C09131=1130.125,26.875,-51.271,179.824,6.474,149.232
C09132=1130.130,26.606,-51.255,179.821,6.473,149.233
C09133=1130.135,26.356,-51.240,179.819,6.472,149.233
C09134=1130.140,26.106,-51.226,179.816,6.471,149.234
C09135=1130.145,25.857,-51.212,179.814,6.470,149.234
C09136=1130.151,25.608,-51.198,179.811,6.469,149.235
C09137=1130.156,25.358,-51.183,179.808,6.468,149.235
C09138=1130.161,25.108,-51.169,179.806,6.467,149.236
C09139=1130.166,24.859,-51.155,179.803,6.465,149.236
C09140=1130.171,24.609,-51.141,179.801,6.465,149.237
C09141=1130.176,24.360,-51.127,179.798,6.463,149.238
C09142=1130.181,24.110,-51.112,179.796,6.462,149.238
C09143=1130.186,23.860,-51.098,179.793,6.462,149.239
C09144=1130.191,23.611,-51.084,179.790,6.460,149.239
C09145=1130.197,23.362,-51.070,179.788,6.460,149.240
C09146=1130.202,23.112,-51.056,179.785,6.458,149.240
C09147=1130.207,22.862,-51.041,179.783,6.458,149.241
C09148=1130.212,22.613,-51.027,179.781,6.457,149.241
C09149=1130.217,22.364,-51.013,179.778,6.455,149.242
C09150=1130.222,22.114,-50.999,179.775,6.455,149.242
C09151=1130.227,21.864,-50.985,179.772,6.453,149.243
C09152=1130.231,21.615,-50.971,179.770,6.452,149.243
C09153=1130.237,21.366,-50.957,179.768,6.452,149.244
C09154=1130.242,21.116,-50.943,179.765,6.450,149.244
C09155=1130.247,20.866,-50.929,179.763,6.449,149.245
C09156=1130.253,20.617,-50.915,179.760,6.448,149.245
C09157=1130.258,20.367,-50.901,179.757,6.447,149.246
C09158=1130.263,20.117,-50.887,179.755,6.447,149.246
C09159=1130.267,19.868,-50.873,179.752,6.445,149.247
C09160=1130.273,19.619,-50.859,179.750,6.445,149.248
C09161=1130.278,19.369,-50.844,179.747,6.443,149.248
C09162=1130.282,19.119,-50.831,179.745,6.442,149.248
C09163=1130.288,18.870,-50.817,179.742,6.442,149.249
C09164=1130.293,18.620,-50.803,179.739,6.440,149.250
C09165=1130.298,18.370,-50.789,179.737,6.439,149.250
C09166=1130.304,18.121,-50.775,179.734,6.438,149.251
C09167=1130.308,17.872,-50.761,179.732,6.437,149.251
C09168=1130.314,17.621,-50.747,179.730,6.436,149.252
C09169=1130.319,17.373,-50.734,179.727,6.435,149.252
C09170=1130.324,17.123,-50.720,179.724,6.434,149.253
C09171=1130.328,16.873,-50.705,179.722,6.434,149.253
C09172=1130.334,16.624,-50.692,179.719,6.432,149.254
C09173=1130.339,16.374,-50.678,179.717,6.432,149.254
C09174=1130.344,16.125,-50.665,179.714,6.430,149.255
C09175=1130.349,15.875,-50.651,179.712,6.429,149.255
C09176=1130.354,15.625,-50.637,179.709,6.429,149.256
C09177=1130.360,15.376,-50.623,179.706,6.427,149.256
C09178=1130.365,15.126,-50.608,179.704,6.426,149.257
C09179=1130.369,14.876,-50.596,179.702,6.425,149.257
C09180=1130.375,14.627,-50.582,179.699,6.424,149.258
C09181=1130.380,14.377,-50.568,179.696,6.423,149.259
C09182=1130.386,14.128,-50.554,179.694,6.423,149.259
C09183=1130.390,13.879,-50.540,179.691,6.421,149.260
C09184=1130.395,13.628,-50.527,179.689,6.421,149.260
C09185=1130.401,13.379,-50.513,179.687,6.420,149.261
C09186=1130.405,13.130,-50.499,179.683,6.419,149.261
C09187=1130.411,12.880,-50.486,179.681,6.418,149.262
C09188=1130.416,12.631,-50.472,179.679,6.417,149.262
C09189=1130.422,12.381,-50.459,179.676,6.416,149.263
C09190=1130.426,12.132,-50.445,179.674,6.415,149.263
C09191=1130.431,11.881,-50.431,179.671,6.414,149.264
C09192=1130.437,11.632,-50.417,179.669,6.413,149.264
C09193=1130.441,11.383,-50.404,179.666,6.412,149.265
C09194=1130.447,11.133,-50.391,179.664,6.411,149.265
C09195=1130.452,10.883,-50.376,179.661,6.410,149.266
C09196=1130.457,10.634,-50.364,179.658,6.409,149.267
C09197=1130.462,10.384,-50.349,179.656,6.408,149.267
C09198=1130.468,10.135,-50.336,179.653,6.407,149.268
C09199=1130.472,9.885,-50.323,179.651,6.406,149.268
C09200=1130.478,9.636,-50.309,179.649,6.406,149.269
C09201=1130.483,9.386,-50.295,179.646,6.404,149.269
C09202=1130.488,9.137,-50.282,179.643,6.404,149.270
C09203=1130.493,8.887,-50.268,179.641,6.403,149.270
C09204=1130.498,8.638,-50.256,179.638,6.401,149.271
C09205=1130.503,8.387,-50.242,179.636,6.400,149.271
C09206=1130.509,8.138,-50.228,179.633,6.400,149.272
C09207=1130.513,7.888,-50.215,179.631,6.398,149.272
C09208=1130.519,7.639,-50.201,179.628,6.398,149.273
C09209=1130.523,7.389,-50.188,179.626,6.397,149.274
C09210=1130.529,7.140,-50.175,179.623,6.396,149.274
C09211=1130.533,6.890,-50.161,179.621,6.395,149.274
C09212=1130.539,6.641,-50.148,179.618,6.394,149.275
C09213=1130.544,6.391,-50.134,179.616,6.394,149.276
C09214=1130.549,6.142,-50.121,179.613,6.392,149.276
C09215=1130.555,5.891,-50.108,179.611,6.392,149.277
C09216=1130.559,5.643,-50.094,179.608,6.391,149.277
C09217=1130.565,5.392,-50.081,179.606,6.389,149.278
C09218=1130.570,5.143,-50.068,179.603,6.388,149.278
C09219=1130.575,4.894,-50.054,179.601,6.388,149.279
C09220=1130.580,4.644,-50.041,179.599,6.387,149.279
C09221=1130.586,4.394,-50.028,179.596,6.386,149.280
C09222=1130.590,4.144,-50.015,179.593,6.385,149.280
C09223=1130.596,3.895,-50.001,179.591,6.384,149.281
C09224=1130.600,3.645,-49.988,179.588,6.383,149.281
C09225=1130.606,3.396,-49.975,179.586,6.382,149.282
C09226=1130.611,3.146,-49.963,179.583,6.382,149.283
C09227=1130.616,2.897,-49.948,179.581,6.381,149.283
C09228=1130.621,2.647,-49.936,179.578,6.380,149.284
C09229=1130.626,2.397,-49.923,179.576,6.379,149.284
C09230=1130.632,2.148,-49.910,179.574,6.378,149.285
C09231=1130.637,1.899,-49.896,179.570,6.377,149.285
C09232=1130.642,1.649,-49.883,179.568,6.376,149.286
C09233=1130.647,1.380,-49.869,179.566,6.375,149.286
C09234=1130.653,1.110,-49.855,179.563,6.374,149.287
C09235=1130.659,0.840,-49.840,179.560,6.373,149.287
C09236=1130.664,0.570,-49.826,179.557,6.372,149.288
C09237=1130.670,0.321,-49.813,179.555,6.371,149.289
C09238=1130.675,0.071,-49.801,179.553,6.370,149.289
C09239=1130.680,-0.179,-49.787,179.550,6.370,149.290
C09240=1130.685,-0.428,-49.774,179.547,6.368,149.290
C09241=1130.690,-0.677,-49.761,179.545,6.367,149.291
C09242=1130.695,-0.927,-49.748,179.543,6.367,149.291
C09243=1130.700,-1.177,-49.735,179.540,6.366,149.292
C09244=1130.705,-1.426,-49.722,179.538,6.365,149.292
C09245=1130.711,-1.676,-49.709,179.535,6.364,149.293
C09246=1130.716,-1.926,-49.696,179.533,6.363,149.293
C09247=1130.721,-2.175,-49.684,179.531,6.363,149.294
C09248=1130.726,-2.425,-49.670,179.528,6.361,149.294
C09249=1130.731,-2.674,-49.657,179.525,6.361,149.295
C09250=1130.736,-2.924,-49.645,179.523,6.360,149.295
C09251=1130.742,-3.174,-49.631,179.521,6.359,149.296
C09252=1130.747,-3.423,-49.619,179.518,6.359,149.297
C09253=1130.752,-3.673,-49.606,179.515,6.357,149.297
C09254=1130.758,-3.922,-49.593,179.513,6.356,149.298
C09255=1130.762,-4.172,-49.580,179.511,6.356,149.298
C09256=1130.767,-4.422,-49.567,179.508,6.355,149.299
C09257=1130.773,-4.671,-49.555,179.506,6.353,149.299
C09258=1130.778,-4.921,-49.541,179.503,6.353,149.300
C09259=1130.783,-5.171,-49.529,179.501,6.352,149.300
C09260=1130.788,-5.420,-49.516,179.499,6.351,149.301
C09261=1130.794,-5.670,-49.503,179.496,6.351,149.301
C09262=1130.798,-5.920,-49.490,179.493,6.349,149.302
C09263=1130.804,-6.169,-49.477,179.491,6.349,149.302
C09264=1130.809,-6.418,-49.465,179.489,6.348,149.303
C09265=1130.814,-6.668,-49.452,179.486,6.347,149.304
C09266=1130.819,-6.918,-49.438,179.484,6.347,149.304
C09267=1130.824,-7.167,-49.426,179.481,6.345,149.305
C09268=1130.830,-7.417,-49.414,179.478,6.345,149.305
C09269=1130.835,-7.666,-49.401,179.476,6.344,149.306
C09270=1130.840,-7.917,-49.388,179.474,6.343,149.306
C09271=1130.845,-8.166,-49.375,179.471,6.342,149.307
C09272=1130.850,-8.415,-49.363,179.469,6.341,149.307
C09273=1130.855,-8.665,-49.350,179.467,6.340,149.308
C09274=1130.860,-8.914,-49.337,179.464,6.340,149.308
C09275=1130.865,-9.165,-49.325,179.462,6.339,149.309
C09276=1130.871,-9.414,-49.312,179.459,6.338,149.309
C09277=1130.876,-9.664,-49.299,179.457,6.337,149.310
C09278=1130.881,-9.913,-49.287,179.454,6.336,149.311
C09279=1130.887,-10.162,-49.274,179.452,6.336,149.311
C09280=1130.891,-10.413,-49.262,179.450,6.335,149.312
C09281=1130.896,-10.662,-49.249,179.447,6.334,149.312
C09282=1130.902,-10.912,-49.237,179.444,6.333,149.313
C09283=1130.907,-11.161,-49.224,179.442,6.332,149.313
C09284=1130.913,-11.411,-49.212,179.439,6.332,149.314
C09285=1130.917,-11.661,-49.199,179.437,6.331,149.314
C09286=1130.923,-11.910,-49.186,179.435,6.330,149.315
C09287=1130.928,-12.160,-49.173,179.433,6.329,149.315
C09288=1130.933,-12.410,-49.162,179.430,6.328,149.316
C09289=1130.938,-12.659,-49.149,179.427,6.327,149.316
C09290=1130.943,-12.908,-49.136,179.425,6.326,149.317
C09291=1130.948,-13.159,-49.124,179.423,6.326,149.318
C09292=1130.953,-13.408,-49.111,179.420,6.325,149.318
C09293=1130.958,-13.658,-49.099,179.418,6.324,149.319
C09294=1130.964,-13.908,-49.087,179.415,6.323,149.319
C09295=1130.969,-14.157,-49.074,179.413,6.322,149.320
C09296=1130.974,-14.406,-49.062,179.411,6.322,149.320
C09297=1130.980,-14.656,-49.050,179.408,6.321,149.321
C09298=1130.985,-14.905,-49.037,179.406,6.320,149.321
C09299=1130.989,-15.155,-49.024,179.404,6.320,149.322
C09300=1130.995,-15.406,-49.012,179.401,6.318,149.322
C09301=1131.000,-15.655,-48.999,179.398,6.318,149.323
C09302=1131.006,-15.905,-48.987,179.396,6.317,149.323
C09303=1131.011,-16.154,-48.975,179.394,6.316,149.324
C09304=1131.016,-16.404,-48.962,179.391,6.316,149.325
C09305=1131.022,-16.654,-48.950,179.389,6.315,149.325
C09306=1131.026,-16.903,-48.938,179.387,6.314,149.326
C09307=1131.031,-17.153,-48.926,179.384,6.313,149.326
C09308=1131.037,-17.402,-48.914,179.381,6.312,149.327
C09309=1131.042,-17.652,-48.902,179.379,6.311,149.327
C09310=1131.046,-17.902,-48.889,179.377,6.311,149.328
C09311=1131.052,-18.152,-48.877,179.374,6.310,149.328
C09312=1131.057,-18.401,-48.864,179.372,6.309,149.329
C09313=1131.062,-18.651,-48.853,179.370,6.309,149.329
C09314=1131.068,-18.900,-48.840,179.367,6.308,149.330
C09315=1131.073,-19.150,-48.828,179.364,6.307,149.330
C09316=1131.078,-19.400,-48.815,179.362,6.306,149.331
C09317=1131.084,-19.649,-48.804,179.360,6.305,149.331
C09318=1131.089,-19.899,-48.791,179.357,6.305,149.332
C09319=1131.094,-20.149,-48.779,179.355,6.304,149.333
C09320=1131.099,-20.398,-48.767,179.353,6.303,149.333
C09321=1131.105,-20.648,-48.755,179.350,6.303,149.334
C09322=1131.109,-20.897,-48.743,179.348,6.302,149.334
C09323=1131.114,-21.147,-48.731,179.345,6.300,149.335
C09324=1131.120,-21.397,-48.719,179.343,6.300,149.335
C09325=1131.125,-21.646,-48.706,179.341,6.299,149.336
C09326=1131.130,-21.896,-48.694,179.338,6.298,149.336
C09327=1131.136,-22.145,-48.682,179.336,6.297,149.337
C09328=1131.141,-22.395,-48.670,179.334,6.297,149.337
C09329=1131.146,-22.645,-48.658,179.331,6.296,149.338
C09330=1131.151,-22.894,-48.646,179.329,6.296,149.338
C09331=1131.156,-23.144,-48.634,179.326,6.295,149.339
C09332=1131.162,-23.394,-48.622,179.324,6.294,149.340
C09333=1131.167,-23.644,-48.610,179.322,6.293,149.340
C09334=1131.172,-23.893,-48.598,179.319,6.292,149.341
C09335=1131.178,-24.143,-48.586,179.317,6.292,149.341
C09336=1131.182,-24.392,-48.574,179.314,6.291,149.342
C09337=1131.189,-24.662,-48.561,179.312,6.290,149.342
C09338=1131.194,-24.933,-48.548,179.310,6.290,149.343
C09339=1131.199,-25.203,-48.535,179.307,6.288,149.343
C09340=1131.205,-25.473,-48.522,179.304,6.288,149.344
C09341=1131.211,-25.723,-48.510,179.302,6.287,149.345
C09342=1131.216,-25.973,-48.498,179.300,6.286,149.345
C09343=1131.221,-26.222,-48.487,179.297,6.286,149.346
C09344=1131.226,-26.472,-48.474,179.295,6.285,149.346
C09345=1131.231,-26.721,-48.463,179.293,6.284,149.347
C09346=1131.237,-26.971,-48.451,179.290,6.284,149.347
C09347=1131.241,-27.221,-48.439,179.288,6.283,149.348
C09348=1131.247,-27.470,-48.427,179.286,6.282,149.348
C09349=1131.252,-27.720,-48.415,179.282,6.281,149.349
C09350=1131.257,-27.970,-48.404,179.280,6.280,149.349
C09351=1131.263,-28.219,-48.392,179.278,6.279,149.350
C09352=1131.268,-28.469,-48.380,179.276,6.279,149.350
C09353=1131.273,-28.718,-48.368,179.273,6.278,149.351
C09354=1131.278,-28.968,-48.356,179.271,6.277,149.352
C09355=1131.283,-29.218,-48.344,179.269,6.277,149.352
C09356=1131.289,-29.468,-48.333,179.267,6.276,149.353
C09357=1131.294,-29.718,-48.321,179.264,6.275,149.353
C09358=1131.299,-29.967,-48.309,179.262,6.275,149.354
C09359=1131.304,-30.217,-48.297,179.260,6.274,149.354
C09360=1131.309,-30.466,-48.286,179.257,6.274,149.355
C09361=1131.315,-30.716,-48.274,179.255,6.273,149.355
C09362=1131.320,-30.966,-48.262,179.253,6.272,149.356
C09363=1131.325,-31.215,-48.251,179.250,6.271,149.356
C09364=1131.330,-31.465,-48.239,179.248,6.271,149.357
C09365=1131.336,-31.715,-48.227,179.246,6.270,149.357
C09366=1131.340,-31.965,-48.216,179.243,6.269,149.358
C09367=1131.346,-32.214,-48.204,179.240,6.268,149.359
C09368=1131.351,-32.464,-48.193,179.238,6.267,149.359
C09369=1131.357,-32.714,-48.181,179.236,6.266,149.360
C09370=1131.362,-32.963,-48.169,179.234,6.266,149.360
C09371=1131.367,-33.213,-48.158,179.231,6.265,149.361
C09372=1131.372,-33.463,-48.146,179.229,6.265,149.361
C09373=1131.377,-33.712,-48.135,179.227,6.264,149.362
C09374=1131.383,-33.962,-48.123,179.224,6.263,149.362
C09375=1131.388,-34.212,-48.111,179.222,6.263,149.363
C09376=1131.393,-34.461,-48.100,179.219,6.262,149.363
C09377=1131.398,-34.711,-48.088,179.217,6.261,149.364
C09378=1131.404,-34.960,-48.077,179.215,6.261,149.365
C09379=1131.409,-35.210,-48.065,179.212,6.260,149.365
C09380=1131.414,-35.460,-48.054,179.210,6.259,149.366
C09381=1131.419,-35.710,-48.042,179.208,6.258,149.366
C09382=1131.425,-35.960,-48.030,179.205,6.258,149.367
C09383=1131.430,-36.209,-48.019,179.203,6.257,149.367
C09384=1131.435,-36.459,-48.007,179.201,6.256,149.368
C09385=1131.440,-36.708,-47.996,179.198,6.256,149.368
C09386=1131.446,-36.958,-47.984,179.196,6.255,149.369
C09387=1131.451,-37.207,-47.973,179.194,6.254,149.369
C09388=1131.456,-37.457,-47.961,179.192,6.254,149.370
C09389=1131.461,-37.707,-47.951,179.189,6.253,149.370
C09390=1131.467,-37.957,-47.939,179.187,6.252,149.371
C09391=1131.472,-38.206,-47.928,179.185,6.252,149.371
C09392=1131.477,-38.456,-47.916,179.183,6.251,149.372
C09393=1131.482,-38.706,-47.905,179.180,6.251,149.373
C09394=1131.488,-38.956,-47.893,179.178,6.250,149.373
C09395=1131.493,-39.205,-47.882,179.176,6.249,149.374
C09396=1131.499,-39.455,-47.871,179.173,6.248,149.374
C09397=1131.503,-39.705,-47.860,179.171,6.248,149.375
C09398=1131.509,-39.955,-47.848,179.168,6.247,149.375
C09399=1131.514,-40.204,-47.837,179.166,6.246,149.376
C09400=1131.519,-40.453,-47.826,179.164,6.246,149.376
C09401=1131.524,-40.704,-47.814,179.161,6.245,149.377
C09402=1131.530,-40.953,-47.803,179.159,6.244,149.377
C09403=1131.535,-41.203,-47.792,179.157,6.244,149.378
C09404=1131.540,-41.452,-47.780,179.154,6.243,149.379
C09405=1131.545,-41.702,-47.768,179.152,6.242,149.379
C09406=1131.551,-41.952,-47.758,179.150,6.242,149.379
C09407=1131.556,-42.201,-47.747,179.148,6.241,149.380
C09408=1131.561,-42.451,-47.735,179.145,6.240,149.381
C09409=1131.567,-42.701,-47.725,179.143,6.240,149.381
C09410=1131.572,-42.951,-47.713,179.141,6.239,149.382
C09411=1131.577,-43.200,-47.702,179.139,6.238,149.382
C09412=1131.582,-43.449,-47.691,179.136,6.238,149.383
C09413=1131.588,-43.700,-47.679,179.134,6.237,149.383
C09414=1131.592,-43.949,-47.668,179.132,6.236,149.384
C09415=1131.598,-44.198,-47.657,179.129,6.235,149.384
C09416=1131.603,-44.449,-47.646,179.127,6.235,149.385
C09417=1131.608,-44.699,-47.635,179.125,6.234,149.385
C09418=1131.613,-44.948,-47.624,179.122,6.233,149.386
C09419=1131.619,-45.198,-47.613,179.121,6.234,149.386
C09420=1131.624,-45.448,-47.601,179.118,6.233,149.387
C09421=1131.629,-45.697,-47.591,179.116,6.232,149.388
C09422=1131.635,-45.947,-47.579,179.114,6.232,149.388
C09423=1131.640,-46.196,-47.568,179.112,6.231,149.388
C09424=1131.645,-46.446,-47.558,179.109,6.230,149.389
C09425=1131.651,-46.696,-47.546,179.107,6.230,149.390
C09426=1131.656,-46.945,-47.535,179.104,6.229,149.390
C09427=1131.661,-47.195,-47.524,179.102,6.228,149.391
C09428=1131.666,-47.445,-47.513,179.100,6.228,149.391
C09429=1131.672,-47.695,-47.502,179.097,6.227,149.392
C09430=1131.677,-47.945,-47.491,179.095,6.226,149.392
C09431=1131.682,-48.193,-47.480,179.093,6.225,149.393
C09432=1131.688,-48.444,-47.469,179.090,6.225,149.393
C09433=1131.692,-48.694,-47.458,179.088,6.224,149.394
C09434=1131.698,-48.943,-47.447,179.086,6.223,149.394
C09435=1131.703,-49.193,-47.436,179.084,6.223,149.395
C09436=1131.709,-49.443,-47.425,179.081,6.222,149.396
C09437=1131.714,-49.692,-47.414,179.080,6.222,149.396
C09438=1131.719,-49.942,-47.404,179.077,6.222,149.397
C09439=1131.724,-50.191,-47.393,179.075,6.221,149.397
C09440=1131.730,-50.442,-47.381,179.072,6.220,149.398
C09441=1131.735,-50.712,-47.370,179.070,6.220,149.398
C09442=1131.741,-50.983,-47.358,179.068,6.219,149.399
C09443=1131.747,-51.254,-47.347,179.065,6.218,149.399
C09444=1131.753,-51.525,-47.334,179.063,6.217,149.400
C09445=1131.758,-51.775,-47.323,179.060,6.217,149.401
C09446=1131.763,-52.024,-47.313,179.058,6.217,149.401
C09447=1131.768,-52.274,-47.302,179.056,6.216,149.402
C09448=1131.774,-52.523,-47.291,179.054,6.215,149.402
C09449=1131.779,-52.773,-47.281,179.052,6.214,149.403
C09450=1131.785,-53.023,-47.269,179.049,6.214,149.403
C09451=1131.790,-53.273,-47.259,179.047,6.213,149.404
C09452=1131.795,-53.522,-47.248,179.045,6.212,149.404
C09453=1131.800,-53.772,-47.237,179.043,6.212,149.405
C09454=1131.805,-54.022,-47.227,179.040,6.211,149.405
C09455=1131.810,-54.271,-47.216,179.038,6.210,149.406
C09456=1131.816,-54.521,-47.206,179.035,6.210,149.406
C09457=1131.821,-54.771,-47.194,179.034,6.210,149.407
C09458=1131.827,-55.020,-47.184,179.031,6.209,149.408
C09459=1131.832,-55.271,-47.173,179.029,6.209,149.408
C09460=1131.836,-55.520,-47.162,179.027,6.208,149.408
C09461=1131.842,-55.770,-47.151,179.025,6.207,149.409
C09462=1131.848,-56.019,-47.141,179.022,6.206,149.409
C09463=1131.853,-56.270,-47.131,179.020,6.206,149.410
C09464=1131.858,-56.518,-47.120,179.018,6.205,149.411
C09465=1131.863,-56.769,-47.109,179.015,6.204,149.411
C09466=1131.869,-57.018,-47.099,179.014,6.204,149.412
C09467=1131.873,-57.268,-47.088,179.011,6.204,149.412
C09468=1131.879,-57.517,-47.077,179.009,6.203,149.413
C09469=1131.885,-57.768,-47.066,179.007,6.202,149.413
C09470=1131.890,-58.017,-47.055,179.005,6.202,149.414
C09471=1131.895,-58.267,-47.045,179.002,6.201,149.414
C09472=1131.900,-58.517,-47.035,179.000,6.201,149.415
C09473=1131.905,-58.767,-47.024,178.998,6.200,149.415
C09474=1131.911,-59.016,-47.014,178.995,6.199,149.416
C09475=1131.916,-59.266,-47.002,178.994,6.199,149.416
C09476=1131.921,-59.516,-46.992,178.991,6.199,149.417
C09477=1131.927,-59.765,-46.982,178.989,6.198,149.418
C09478=1131.932,-60.015,-46.972,178.987,6.197,149.418
C09479=1131.937,-60.264,-46.961,178.985,6.196,149.418
C09480=1131.942,-60.515,-46.950,178.982,6.196,149.419
C09481=1131.948,-60.764,-46.940,178.980,6.195,149.420
C09482=1131.953,-61.014,-46.929,178.978,6.195,149.420
C09483=1131.958,-61.264,-46.919,178.976,6.195,149.421
C09484=1131.964,-61.513,-46.909,178.974,6.194,149.421
C09485=1131.969,-61.763,-46.898,178.971,6.193,149.422
C09486=1131.974,-62.013,-46.887,178.969,6.193,149.422
C09487=1131.979,-62.263,-46.877,178.967,6.192,149.423
C09488=1131.985,-62.512,-46.867,178.964,6.191,149.423
C09489=1131.990,-62.762,-46.857,178.963,6.191,149.424
C09490=1131.995,-63.012,-46.846,178.961,6.190,149.424
C09491=1132.000,-63.261,-46.836,178.958,6.190,149.425
C09492=1132.005,-63.512,-46.826,178.956,6.189,149.425
C09493=1132.011,-63.761,-46.815,178.954,6.188,149.426
C09494=1132.016,-64.010,-46.804,178.951,6.188,149.426
C09495=1132.021,-64.260,-46.794,178.949,6.187,149.427
C09496=1132.027,-64.510,-46.784,178.947,6.187,149.428
C09497=1132.032,-64.759,-46.773,178.945,6.187,149.428
C09498=1132.037,-65.010,-46.763,178.943,6.186,149.429
C09499=1132.043,-65.259,-46.753,178.941,6.185,149.429
C09500=1132.049,-65.509,-46.742,178.938,6.184,149.429
C09501=1132.054,-65.759,-46.732,178.936,6.184,149.430
C09502=1132.058,-66.008,-46.722,178.934,6.184,149.431
C09503=1132.063,-66.259,-46.712,178.932,6.183,149.431
C09504=1132.069,-66.508,-46.701,178.930,6.182,149.432
C09505=1132.075,-66.758,-46.691,178.928,6.182,149.432
C09506=1132.080,-67.008,-46.681,178.925,6.181,149.433
C09507=1132.085,-67.257,-46.670,178.923,6.181,149.433
C09508=1132.091,-67.507,-46.660,178.921,6.181,149.434
C09509=1132.096,-67.756,-46.651,178.919,6.180,149.434
C09510=1132.101,-68.006,-46.640,178.917,6.179,149.435
C09511=1132.106,-68.256,-46.630,178.914,6.179,149.435
C09512=1132.112,-68.505,-46.620,178.912,6.178,149.436
C09513=1132.117,-68.756,-46.609,178.910,6.177,149.436
C09514=1132.123,-69.005,-46.599,178.908,6.177,149.437
C09515=1132.127,-69.255,-46.589,178.906,6.176,149.437
C09516=1132.132,-69.505,-46.579,178.904,6.176,149.438
C09517=1132.138,-69.754,-46.568,178.901,6.175,149.439
C09518=1132.144,-70.004,-46.559,178.899,6.175,149.439
C09519=1132.149,-70.254,-46.549,178.897,6.175,149.440
C09520=1132.154,-70.504,-46.538,178.895,6.174,149.440
C09521=1132.159,-70.753,-46.529,178.893,6.173,149.441
C09522=1132.165,-71.003,-46.518,178.890,6.173,149.441
C09523=1132.171,-71.253,-46.508,178.888,6.172,149.442
C09524=1132.176,-71.503,-46.498,178.886,6.172,149.442
C09525=1132.180,-71.752,-46.488,178.884,6.171,149.443
C09526=1132.186,-72.002,-46.478,178.882,6.170,149.443
C09527=1132.191,-72.252,-46.468,178.880,6.170,149.444
C09528=1132.197,-72.502,-46.458,178.877,6.169,149.444
C09529=1132.202,-72.751,-46.448,178.876,6.169,149.445
C09530=1132.207,-73.001,-46.438,178.873,6.169,149.445
C09531=1132.213,-73.250,-46.428,178.871,6.168,149.446
C09532=1132.218,-73.501,-46.418,178.869,6.167,149.446
C09533=1132.223,-73.750,-46.408,178.867,6.166,149.447
C09534=1132.229,-74.000,-46.398,178.865,6.167,149.447
C09535=1132.234,-74.249,-46.388,178.862,6.166,149.448
C09536=1132.239,-74.500,-46.377,178.860,6.165,149.448
C09537=1132.244,-74.750,-46.368,178.858,6.164,149.449
C09538=1132.250,-74.999,-46.358,178.856,6.164,149.449
C09539=1132.256,-75.249,-46.348,178.854,6.164,149.450
C09540=1132.261,-75.498,-46.338,178.852,6.163,149.451
C09541=1132.266,-75.749,-46.328,178.849,6.163,149.451
C09542=1132.271,-75.998,-46.318,178.847,6.162,149.452
C09543=1132.277,-76.248,-46.308,178.846,6.162,149.452
C09544=1132.282,-76.497,-46.298,178.843,6.161,149.453
C09545=1132.288,-76.769,-46.288,178.841,6.161,149.453
C09546=1132.293,-77.041,-46.277,178.839,6.160,149.454
C09547=1132.299,-77.312,-46.267,178.836,6.159,149.454
C09548=1132.305,-77.583,-46.255,178.834,6.159,149.455
C09549=1132.310,-77.833,-46.246,178.831,6.158,149.455
C09550=1132.316,-78.083,-46.236,178.830,6.158,149.456
C09551=1132.321,-78.333,-46.226,178.828,6.157,149.456
C09552=1132.326,-78.583,-46.217,178.826,6.157,149.457
C09553=1132.332,-78.832,-46.206,178.823,6.156,149.457
C09554=1132.337,-79.082,-46.196,178.821,6.155,149.458
C09555=1132.343,-79.332,-46.187,178.819,6.156,149.459
C09556=1132.348,-79.581,-46.177,178.817,6.155,149.459
C09557=1132.354,-79.831,-46.167,178.815,6.154,149.459
C09558=1132.358,-80.082,-46.158,178.812,6.153,149.460
C09559=1132.364,-80.331,-46.147,178.811,6.153,149.460
C09560=1132.369,-80.581,-46.139,178.809,6.153,149.461
C09561=1132.375,-80.830,-46.128,178.806,6.152,149.461
C09562=1132.380,-81.080,-46.119,178.804,6.151,149.462
C09563=1132.385,-81.330,-46.109,178.802,6.151,149.463
C09564=1132.391,-81.579,-46.099,178.800,6.151,149.463
C09565=1132.396,-81.829,-46.090,178.798,6.150,149.464
C09566=1132.401,-82.079,-46.080,178.796,6.149,149.464
C09567=1132.406,-82.329,-46.071,178.794,6.149,149.465
C09568=1132.412,-82.579,-46.060,178.792,6.148,149.465
C09569=1132.417,-82.828,-46.051,178.789,6.148,149.466
C09570=1132.423,-83.078,-46.041,178.787,6.147,149.466
C09571=1132.428,-83.327,-46.032,178.785,6.147,149.467
C09572=1132.434,-83.578,-46.022,178.783,6.147,149.467
C09573=1132.439,-83.827,-46.012,178.781,6.146,149.468
C09574=1132.444,-84.077,-46.003,178.779,6.146,149.468
C09575=1132.449,-84.327,-45.993,178.777,6.145,149.469
C09576=1132.454,-84.577,-45.984,178.775,6.144,149.469
C09577=1132.460,-84.827,-45.973,178.772,6.144,149.470
C09578=1132.465,-85.077,-45.965,178.771,6.144,149.470
C09579=1132.471,-85.326,-45.954,178.769,6.143,149.471
C09580=1132.476,-85.576,-45.945,178.766,6.143,149.471
C09581=1132.481,-85.825,-45.936,178.764,6.142,149.472
C09582=1132.487,-86.075,-45.926,178.763,6.142,149.472
C09583=1132.492,-86.325,-45.917,178.760,6.141,149.473
C09584=1132.498,-86.575,-45.907,178.758,6.140,149.473
C09585=1132.503,-86.825,-45.898,178.756,6.141,149.474
C09586=1132.508,-87.074,-45.888,178.754,6.140,149.474
C09587=1132.513,-87.324,-45.879,178.752,6.139,149.475
C09588=1132.519,-87.574,-45.869,178.750,6.138,149.475
C09589=1132.524,-87.823,-45.860,178.748,6.139,149.476
C09590=1132.529,-88.074,-45.850,178.746,6.138,149.476
C09591=1132.534,-88.323,-45.841,178.744,6.137,149.477
C09592=1132.540,-88.573,-45.832,178.742,6.137,149.477
C09593=1132.545,-88.823,-45.822,178.740,6.136,149.478
C09594=1132.550,-89.073,-45.813,178.737,6.136,149.479
C09595=1132.556,-89.322,-45.802,178.735,6.135,149.479
C09596=1132.561,-89.572,-45.794,178.733,6.135,149.479
C09597=1132.566,-89.822,-45.785,178.731,6.134,149.480
C09598=1132.572,-90.072,-45.774,178.729,6.134,149.480
C09599=1132.577,-90.321,-45.766,178.727,6.134,149.481
C09600=1132.583,-90.572,-45.756,178.725,6.133,149.481
C09601=1132.588,-90.821,-45.746,178.723,6.132,149.482
C09602=1132.593,-91.071,-45.738,178.721,6.132,149.482
C09603=1132.599,-91.321,-45.728,178.719,6.132,149.483
C09604=1132.604,-91.570,-45.718,178.717,6.131,149.483
C09605=1132.609,-91.820,-45.710,178.715,6.131,149.484
C09606=1132.615,-92.070,-45.700,178.713,6.130,149.485
C09607=1132.620,-92.320,-45.691,178.710,6.130,149.485
C09608=1132.626,-92.569,-45.681,178.708,6.129,149.486
C09609=1132.631,-92.819,-45.672,178.707,6.129,149.486
C09610=1132.636,-93.069,-45.663,178.704,6.128,149.487
C09611=1132.641,-93.319,-45.653,178.702,6.128,149.487
C09612=1132.647,-93.569,-45.644,178.701,6.128,149.487
C09613=1132.652,-93.818,-45.635,178.698,6.127,149.488
C09614=1132.658,-94.068,-45.626,178.696,6.126,149.488
C09615=1132.663,-94.317,-45.616,178.695,6.126,149.489
C09616=1132.668,-94.567,-45.607,178.692,6.126,149.490
C09617=1132.674,-94.817,-45.598,178.690,6.125,149.490
C09618=1132.679,-95.067,-45.589,178.688,6.125,149.491
C09619=1132.685,-95.317,-45.580,178.686,6.124,149.491
C09620=1132.689,-95.566,-45.571,178.684,6.124,149.492
C09621=1132.695,-95.816,-45.561,178.682,6.124,149.492
C09622=1132.701,-96.066,-45.552,178.680,6.123,149.493
C09623=1132.706,-96.316,-45.543,178.678,6.122,149.493
C09624=1132.712,-96.566,-45.534,178.676,6.122,149.494
C09625=1132.716,-96.815,-45.524,178.674,6.121,149.494
C09626=1132.722,-97.065,-45.515,178.672,6.121,149.495
C09627=1132.727,-97.315,-45.506,178.670,6.121,149.495
C09628=1132.733,-97.564,-45.497,178.668,6.120,149.495
C09629=1132.738,-97.814,-45.488,178.666,6.119,149.496
C09630=1132.744,-98.064,-45.479,178.664,6.120,149.497
C09631=1132.749,-98.314,-45.471,178.662,6.119,149.497
C09632=1132.754,-98.564,-45.460,178.659,6.118,149.498
C09633=1132.760,-98.813,-45.451,178.658,6.118,149.498
C09634=1132.765,-99.063,-45.443,178.656,6.117,149.499
C09635=1132.770,-99.313,-45.434,178.653,6.117,149.499
C09636=1132.776,-99.563,-45.424,178.652,6.117,149.500
C09637=1132.782,-99.812,-45.416,178.650,6.116,149.500
C09638=1132.787,-100.062,-45.407,178.647,6.115,149.501
C09639=1132.792,-100.312,-45.398,178.646,6.115,149.501
C09640=1132.797,-100.562,-45.389,178.644,6.114,149.502
C09641=1132.803,-100.812,-45.379,178.641,6.114,149.502
C09642=1132.808,-101.062,-45.371,178.640,6.114,149.503
C09643=1132.813,-101.312,-45.362,178.638,6.113,149.503
C09644=1132.818,-101.562,-45.353,178.636,6.113,149.503
C09645=1132.824,-101.810,-45.344,178.634,6.112,149.504
C09646=1132.829,-102.060,-45.335,178.632,6.112,149.504
C09647=1132.835,-102.310,-45.325,178.630,6.112,149.505
C09648=1132.840,-102.560,-45.316,178.628,6.111,149.505
C09649=1132.846,-102.833,-45.307,178.625,6.111,149.506
C09650=1132.852,-103.105,-45.297,178.623,6.110,149.507
C09651=1132.857,-103.377,-45.287,178.621,6.110,149.507
C09652=1132.864,-103.649,-45.278,178.619,6.109,149.508
C09653=1132.869,-103.899,-45.269,178.617,6.108,149.508
C09654=1132.874,-104.149,-45.260,178.615,6.108,149.509
C09655=1132.879,-104.398,-45.251,178.613,6.108,149.509
C09656=1132.885,-104.649,-45.242,178.611,6.107,149.510
C09657=1132.890,-104.898,-45.233,178.609,6.107,149.510
C09658=1132.896,-105.148,-45.224,178.607,6.107,149.511
C09659=1132.901,-105.397,-45.215,178.605,6.107,149.511
C09660=1132.906,-105.647,-45.206,178.603,6.106,149.512
C09661=1132.912,-105.898,-45.198,178.601,6.105,149.512
C09662=1132.917,-106.148,-45.189,178.599,6.105,149.513
C09663=1132.923,-106.397,-45.181,178.597,6.104,149.513
C09664=1132.928,-106.647,-45.172,178.595,6.104,149.514
C09665=1132.933,-106.897,-45.163,178.593,6.104,149.514
C09666=1132.938,-107.146,-45.154,178.591,6.103,149.515
C09667=1132.943,-107.396,-45.145,178.589,6.103,149.515
C09668=1132.950,-107.646,-45.136,178.587,6.102,149.516
C09669=1132.955,-107.896,-45.127,178.585,6.102,149.516
C09670=1132.960,-108.145,-45.118,178.583,6.102,149.517
C09671=1132.966,-108.396,-45.110,178.581,6.101,149.517
C09672=1132.971,-108.645,-45.102,178.580,6.101,149.518
C09673=1132.977,-108.895,-45.093,178.577,6.100,149.518
C09674=1132.982,-109.145,-45.084,178.575,6.099,149.519
C09675=1132.987,-109.395,-45.075,178.574,6.099,149.519
C09676=1132.992,-109.644,-45.066,178.571,6.099,149.520
C09677=1132.998,-109.894,-45.057,178.570,6.099,149.520
C09678=1133.003,-110.144,-45.049,178.568,6.098,149.520
C09679=1133.009,-110.394,-45.040,178.565,6.097,149.521
C09680=1133.014,-110.644,-45.031,178.564,6.097,149.521
C09681=1133.019,-110.893,-45.023,178.562,6.097,149.522
C09682=1133.025,-111.143,-45.014,178.560,6.097,149.522
C09683=1133.030,-111.393,-45.006,178.558,6.096,149.523
C09684=1133.036,-111.642,-44.997,178.556,6.095,149.523
C09685=1133.041,-111.892,-44.988,178.554,6.095,149.524
C09686=1133.046,-112.142,-44.980,178.552,6.094,149.524
C09687=1133.051,-112.392,-44.971,178.550,6.094,149.525
C09688=1133.057,-112.642,-44.963,178.548,6.094,149.525
C09689=1133.063,-112.892,-44.954,178.546,6.094,149.526
C09690=1133.068,-113.141,-44.945,178.544,6.093,149.526
C09691=1133.074,-113.391,-44.936,178.542,6.092,149.527
C09692=1133.079,-113.641,-44.928,178.540,6.092,149.527
C09693=1133.084,-113.891,-44.919,178.538,6.092,149.528
C09694=1133.089,-114.141,-44.911,178.537,6.092,149.528
C09695=1133.095,-114.390,-44.903,178.534,6.091,149.529
C09696=1133.100,-114.640,-44.894,178.532,6.090,149.529
C09697=1133.105,-114.890,-44.885,178.531,6.090,149.530
C09698=1133.111,-115.139,-44.877,178.528,6.089,149.530
C09699=1133.116,-115.389,-44.869,178.527,6.089,149.531
C09700=1133.121,-115.639,-44.860,178.525,6.089,149.531
C09701=1133.127,-115.888,-44.851,178.523,6.089,149.532
C09702=1133.133,-116.139,-44.843,178.521,6.088,149.532
C09703=1133.138,-116.389,-44.834,178.519,6.087,149.533
C09704=1133.144,-116.638,-44.826,178.517,6.087,149.533
C09705=1133.149,-116.888,-44.818,178.515,6.086,149.533
C09706=1133.154,-117.138,-44.809,178.514,6.086,149.534
C09707=1133.160,-117.387,-44.800,178.512,6.085,149.534
C09708=1133.165,-117.638,-44.793,178.510,6.086,149.535
C09709=1133.170,-117.887,-44.784,178.508,6.085,149.535
C09710=1133.176,-118.137,-44.776,178.506,6.085,149.536
C09711=1133.181,-118.387,-44.767,178.504,6.084,149.536
C09712=1133.186,-118.637,-44.758,178.502,6.083,149.537
C09713=1133.192,-118.887,-44.750,178.500,6.083,149.537
C09714=1133.198,-119.137,-44.741,178.498,6.083,149.538
C09715=1133.202,-119.387,-44.734,178.496,6.083,149.538
C09716=1133.208,-119.636,-44.725,178.494,6.082,149.539
C09717=1133.213,-119.886,-44.716,178.493,6.082,149.539
C09718=1133.219,-120.135,-44.708,178.490,6.081,149.540
C09719=1133.224,-120.385,-44.700,178.489,6.081,149.540
C09720=1133.230,-120.636,-44.691,178.487,6.081,149.541
C09721=1133.235,-120.885,-44.683,178.484,6.080,149.541
C09722=1133.240,-121.135,-44.675,178.483,6.080,149.542
C09723=1133.246,-121.385,-44.666,178.481,6.079,149.542
C09724=1133.252,-121.635,-44.659,178.479,6.079,149.543
C09725=1133.257,-121.885,-44.650,178.477,6.078,149.543
C09726=1133.262,-122.133,-44.642,178.476,6.078,149.543
C09727=1133.267,-122.384,-44.634,178.473,6.077,149.544
C09728=1133.273,-122.634,-44.625,178.472,6.077,149.544
C09729=1133.279,-122.883,-44.617,178.470,6.077,149.545
C09730=1133.284,-123.133,-44.608,178.468,6.077,149.545
C09731=1133.289,-123.383,-44.601,178.466,6.076,149.546
C09732=1133.294,-123.633,-44.592,178.464,6.076,149.546
C09733=1133.300,-123.882,-44.584,178.462,6.075,149.547
C09734=1133.305,-124.132,-44.575,178.461,6.075,149.547
C09735=1133.310,-124.382,-44.568,178.458,6.075,149.548
C09736=1133.316,-124.632,-44.560,178.456,6.074,149.548
C09737=1133.321,-124.882,-44.551,178.455,6.074,149.549
C09738=1133.328,-125.132,-44.543,178.452,6.073,149.549
C09739=1133.332,-125.381,-44.535,178.451,6.073,149.550
C09740=1133.338,-125.631,-44.527,178.449,6.072,149.550
C09741=1133.343,-125.881,-44.518,178.447,6.072,149.551
C09742=1133.349,-126.131,-44.510,178.445,6.071,149.551
C09743=1133.354,-126.380,-44.502,178.444,6.071,149.551
C09744=1133.359,-126.631,-44.494,178.441,6.071,149.552
C09745=1133.365,-126.881,-44.486,178.440,6.071,149.552
C09746=1133.370,-127.130,-44.478,178.438,6.070,149.553
C09747=1133.376,-127.380,-44.470,178.436,6.070,149.553
C09748=1133.381,-127.630,-44.461,178.434,6.069,149.554
C09749=1133.387,-127.879,-44.453,178.432,6.069,149.554
C09750=1133.392,-128.130,-44.445,178.430,6.068,149.555
C09751=1133.398,-128.379,-44.437,178.429,6.068,149.555
C09752=1133.403,-128.629,-44.429,178.427,6.068,149.556
C09753=1132.982,-128.640,-44.473,178.423,6.072,149.557
C09754=1132.976,-128.390,-44.481,178.425,6.072,149.557
C09755=1132.971,-128.141,-44.490,178.427,6.072,149.556
C09756=1132.966,-127.891,-44.497,178.429,6.072,149.556
C09757=1132.960,-127.641,-44.506,178.431,6.073,149.556
C09758=1132.955,-127.391,-44.514,178.433,6.073,149.555
C09759=1132.949,-127.141,-44.521,178.435,6.074,149.555
C09760=1132.944,-126.892,-44.530,178.436,6.074,149.554
C09761=1132.938,-126.642,-44.538,178.438,6.075,149.554
C09762=1132.934,-126.392,-44.546,178.440,6.075,149.553
C09763=1132.928,-126.143,-44.554,178.442,6.075,149.553
C09764=1132.922,-125.892,-44.562,178.444,6.075,149.552
C09765=1132.917,-125.642,-44.571,178.446,6.076,149.552
C09766=1132.912,-125.393,-44.578,178.447,6.076,149.551
C09767=1132.906,-125.143,-44.587,178.450,6.077,149.551
C09768=1132.900,-124.893,-44.595,178.452,6.078,149.550
C09769=1132.895,-124.643,-44.604,178.453,6.078,149.550
C09770=1132.890,-124.394,-44.611,178.456,6.078,149.549
C09771=1132.885,-124.144,-44.620,178.457,6.079,149.549
C09772=1132.879,-123.894,-44.628,178.459,6.079,149.549
C09773=1132.873,-123.644,-44.637,178.460,6.079,149.548
C09774=1132.869,-123.394,-44.644,178.463,6.080,149.548
C09775=1132.863,-123.144,-44.652,178.464,6.080,149.547
C09776=1132.858,-122.895,-44.661,178.466,6.081,149.547
C09777=1132.851,-122.645,-44.669,178.468,6.081,149.546
C09778=1132.846,-122.395,-44.678,178.470,6.081,149.546
C09779=1132.842,-122.145,-44.686,178.472,6.081,149.545
C09780=1132.836,-121.896,-44.694,178.474,6.082,149.545
C09781=1132.831,-121.646,-44.703,178.476,6.082,149.544
C09782=1132.825,-121.396,-44.711,178.478,6.083,149.544
C09783=1132.820,-121.147,-44.719,178.480,6.084,149.543
C09784=1132.815,-120.896,-44.727,178.482,6.084,149.543
C09785=1132.809,-120.647,-44.736,178.483,6.085,149.543
C09786=1132.803,-120.396,-44.744,178.485,6.085,149.542
C09787=1132.798,-120.147,-44.753,178.487,6.085,149.542
C09788=1132.792,-119.897,-44.760,178.489,6.085,149.541
C09789=1132.788,-119.647,-44.769,178.491,6.086,149.541
C09790=1132.782,-119.398,-44.777,178.493,6.086,149.540
C09791=1132.776,-119.148,-44.785,178.495,6.087,149.540
C09792=1132.771,-118.898,-44.794,178.496,6.087,149.539
C09793=1132.765,-118.648,-44.802,178.499,6.087,149.539
C09794=1132.760,-118.398,-44.811,178.501,6.088,149.538
C09795=1132.755,-118.148,-44.820,178.502,6.088,149.538
C09796=1132.750,-117.899,-44.827,178.505,6.089,149.537
C09797=1132.744,-117.649,-44.836,178.506,6.089,149.537
C09798=1132.739,-117.399,-44.844,178.508,6.090,149.536
C09799=1132.733,-117.149,-44.853,178.510,6.090,149.536
C09800=1132.728,-116.900,-44.862,178.512,6.090,149.535
C09801=1132.723,-116.649,-44.870,178.514,6.090,149.535
C09802=1132.717,-116.400,-44.878,178.516,6.091,149.534
C09803=1132.712,-116.150,-44.887,178.518,6.092,149.534
C09804=1132.706,-115.900,-44.895,178.520,6.092,149.533
C09805=1132.701,-115.651,-44.903,178.522,6.092,149.533
C09806=1132.696,-115.401,-44.912,178.523,6.093,149.533
C09807=1132.690,-115.150,-44.921,178.525,6.093,149.532
C09808=1132.685,-114.901,-44.929,178.527,6.093,149.532
C09809=1132.680,-114.651,-44.938,178.529,6.094,149.531
C09810=1132.674,-114.402,-44.947,178.531,6.095,149.531
C09811=1132.668,-114.152,-44.955,178.533,6.095,149.530
C09812=1132.663,-113.902,-44.964,178.535,6.096,149.530
C09813=1132.658,-113.652,-44.972,178.537,6.096,149.529
C09814=1132.652,-113.402,-44.980,178.539,6.096,149.529
C09815=1132.647,-113.152,-44.989,178.541,6.097,149.528
C09816=1132.642,-112.903,-44.998,178.543,6.097,149.528
C09817=1132.636,-112.653,-45.007,178.545,6.098,149.527
C09818=1132.630,-112.403,-45.015,178.546,6.098,149.527
C09819=1132.625,-112.153,-45.024,178.549,6.098,149.526
C09820=1132.620,-111.903,-45.033,178.550,6.098,149.526
C09821=1132.614,-111.654,-45.041,178.552,6.099,149.525
C09822=1132.609,-111.404,-45.049,178.555,6.100,149.525
C09823=1132.604,-111.154,-45.058,178.556,6.100,149.524
C09824=1132.598,-110.904,-45.067,178.558,6.101,149.524
C09825=1132.593,-110.655,-45.076,178.560,6.101,149.523
C09826=1132.587,-110.405,-45.085,178.562,6.101,149.523
C09827=1132.582,-110.155,-45.093,178.564,6.102,149.522
C09828=1132.577,-109.905,-45.102,178.566,6.102,149.522
C09829=1132.571,-109.656,-45.110,178.568,6.103,149.521
C09830=1132.566,-109.406,-45.119,178.570,6.103,149.521
C09831=1132.561,-109.156,-45.128,178.572,6.103,149.520
C09832=1132.556,-108.906,-45.137,178.574,6.104,149.520
C09833=1132.550,-108.657,-45.145,178.576,6.104,149.519
C09834=1132.544,-108.406,-45.154,178.578,6.105,149.519
C09835=1132.539,-108.156,-45.162,178.580,6.105,149.518
C09836=1132.534,-107.907,-45.171,178.582,6.106,149.518
C09837=1132.528,-107.657,-45.180,178.584,6.106,149.517
C09838=1132.523,-107.408,-45.189,178.586,6.106,149.517
C09839=1132.518,-107.158,-45.198,178.588,6.107,149.516
C09840=1132.513,-106.908,-45.207,178.589,6.107,149.516
C09841=1132.508,-106.658,-45.215,178.592,6.108,149.515
C09842=1132.501,-106.408,-45.223,178.594,6.108,149.515
C09843=1132.496,-106.158,-45.232,178.595,6.108,149.515
C09844=1132.490,-105.908,-45.242,178.598,6.109,149.514
C09845=1132.485,-105.658,-45.251,178.600,6.110,149.514
C09846=1132.480,-105.409,-45.259,178.601,6.110,149.513
C09847=1132.474,-105.159,-45.268,178.604,6.111,149.513
C09848=1132.469,-104.910,-45.277,178.605,6.111,149.512
C09849=1132.464,-104.660,-45.286,178.607,6.111,149.512
C09850=1132.459,-104.410,-45.295,178.610,6.112,149.511
C09851=1132.454,-104.160,-45.304,178.611,6.112,149.511
C09852=1132.448,-103.910,-45.312,178.614,6.112,149.510
C09853=1132.442,-103.661,-45.322,178.616,6.113,149.509
C09854=1132.436,-103.388,-45.331,178.618,6.113,149.509
C09855=1132.431,-103.116,-45.341,178.620,6.114,149.508
C09856=1132.425,-102.844,-45.351,178.622,6.115,149.508
C09857=1132.419,-102.571,-45.360,178.624,6.115,149.507
C09858=1132.414,-102.321,-45.369,178.626,6.115,149.507
C09859=1132.409,-102.071,-45.378,178.628,6.116,149.506
C09860=1132.403,-101.822,-45.387,178.631,6.116,149.506
C09861=1132.398,-101.572,-45.396,178.632,6.116,149.505
C09862=1132.392,-101.322,-45.405,178.634,6.117,149.505
C09863=1132.387,-101.072,-45.414,178.636,6.117,149.504
C09864=1132.382,-100.823,-45.423,178.638,6.118,149.504
C09865=1132.376,-100.573,-45.432,178.640,6.119,149.503
C09866=1132.372,-100.324,-45.441,178.642,6.118,149.503
C09867=1132.365,-100.074,-45.451,178.644,6.119,149.502
C09868=1132.360,-99.824,-45.459,178.646,6.120,149.502
C09869=1132.355,-99.574,-45.468,178.648,6.120,149.501
C09870=1132.350,-99.324,-45.477,178.650,6.121,149.501
C09871=1132.344,-99.075,-45.486,178.652,6.121,149.500
C09872=1132.338,-98.824,-45.496,178.654,6.121,149.500
C09873=1132.333,-98.575,-45.504,178.656,6.122,149.499
C09874=1132.328,-98.325,-45.513,178.658,6.123,149.499
C09875=1132.323,-98.075,-45.522,178.660,6.123,149.498
C09876=1132.317,-97.826,-45.532,178.662,6.124,149.498
C09877=1132.312,-97.576,-45.541,178.664,6.124,149.498
C09878=1132.306,-97.326,-45.550,178.666,6.124,149.497
C09879=1132.301,-97.077,-45.559,178.669,6.125,149.496
C09880=1132.295,-96.826,-45.568,178.671,6.125,149.496
C09881=1132.290,-96.577,-45.577,178.672,6.125,149.495
C09882=1132.285,-96.327,-45.586,178.675,6.126,149.495
C09883=1132.279,-96.077,-45.596,178.677,6.127,149.494
C09884=1132.274,-95.827,-45.605,178.678,6.127,149.494
C09885=1132.269,-95.577,-45.614,178.681,6.128,149.493
C09886=1132.264,-95.328,-45.623,178.683,6.128,149.493
C09887=1132.258,-95.077,-45.633,178.684,6.128,149.492
C09888=1132.253,-94.829,-45.642,178.687,6.129,149.492
C09889=1132.247,-94.579,-45.651,178.689,6.130,149.491
C09890=1132.242,-94.329,-45.660,178.690,6.130,149.491
C09891=1132.236,-94.079,-45.669,178.693,6.130,149.490
C09892=1132.231,-93.830,-45.679,178.695,6.131,149.490
C09893=1132.226,-93.580,-45.688,178.697,6.131,149.489
C09894=1132.220,-93.330,-45.697,178.699,6.132,149.489
C09895=1132.215,-93.080,-45.706,178.701,6.132,149.488
C09896=1132.210,-92.830,-45.716,178.703,6.132,149.488
C09897=1132.204,-92.581,-45.725,178.705,6.133,149.487
C09898=1132.199,-92.331,-45.734,178.707,6.134,149.487
C09899=1132.193,-92.081,-45.743,178.709,6.134,149.486
C09900=1132.189,-91.831,-45.753,178.711,6.134,149.486
C09901=1132.183,-91.581,-45.762,178.713,6.135,149.485
C09902=1132.177,-91.331,-45.771,178.715,6.136,149.485
C09903=1132.173,-91.082,-45.781,178.717,6.136,149.484
C09904=1132.167,-90.832,-45.790,178.720,6.136,149.484
C09905=1132.162,-90.582,-45.799,178.722,6.137,149.483
C09906=1132.157,-90.333,-45.809,178.723,6.137,149.483
C09907=1132.151,-90.083,-45.819,178.726,6.138,149.482
C09908=1132.146,-89.833,-45.827,178.728,6.139,149.482
C09909=1132.141,-89.584,-45.837,178.729,6.138,149.481
C09910=1132.135,-89.333,-45.847,178.732,6.139,149.481
C09911=1132.130,-89.084,-45.855,178.734,6.140,149.480
C09912=1132.124,-88.834,-45.866,178.736,6.141,149.480
C09913=1132.119,-88.584,-45.875,178.738,6.141,149.479
C09914=1132.114,-88.335,-45.884,178.740,6.141,149.479
C09915=1132.108,-88.085,-45.894,178.743,6.142,149.478
C09916=1132.103,-87.835,-45.903,178.744,6.142,149.478
C09917=1132.097,-87.585,-45.913,178.746,6.143,149.477
C09918=1132.092,-87.335,-45.922,178.749,6.143,149.477
C09919=1132.087,-87.086,-45.932,178.751,6.144,149.476
C09920=1132.081,-86.836,-45.941,178.752,6.144,149.476
C09921=1132.076,-86.586,-45.950,178.754,6.145,149.475
C09922=1132.071,-86.336,-45.960,178.757,6.146,149.475
C09923=1132.066,-86.086,-45.969,178.758,6.145,149.474
C09924=1132.061,-85.837,-45.979,178.761,6.146,149.474
C09925=1132.055,-85.587,-45.988,178.763,6.147,149.473
C09926=1132.050,-85.337,-45.998,178.765,6.147,149.473
C09927=1132.045,-85.087,-46.007,178.767,6.147,149.472
C09928=1132.039,-84.838,-46.018,178.769,6.148,149.472
C09929=1132.034,-84.588,-46.026,178.771,6.149,149.471
C09930=1132.028,-84.338,-46.037,178.773,6.149,149.471
C09931=1132.023,-84.089,-46.046,178.775,6.150,149.470
C09932=1132.017,-83.839,-46.056,178.778,6.150,149.469
C09933=1132.012,-83.589,-46.065,178.780,6.151,149.469
C09934=1132.007,-83.339,-46.075,178.782,6.151,149.469
C09935=1132.002,-83.089,-46.084,178.784,6.151,149.468
C09936=1131.997,-82.840,-46.094,178.786,6.152,149.468
C09937=1131.991,-82.590,-46.103,178.788,6.153,149.467
C09938=1131.986,-82.340,-46.113,178.790,6.153,149.467
C09939=1131.980,-82.090,-46.123,178.792,6.154,149.466
C09940=1131.975,-81.841,-46.133,178.795,6.154,149.465
C09941=1131.969,-81.591,-46.143,178.797,6.155,149.465
C09942=1131.964,-81.341,-46.152,178.798,6.155,149.464
C09943=1131.959,-81.091,-46.162,178.801,6.155,149.464
C09944=1131.954,-80.841,-46.171,178.803,6.156,149.463
C09945=1131.948,-80.592,-46.181,178.805,6.157,149.463
C09946=1131.943,-80.342,-46.192,178.807,6.157,149.462
C09947=1131.938,-80.092,-46.200,178.809,6.158,149.462
C09948=1131.932,-79.843,-46.211,178.811,6.158,149.461
C09949=1131.927,-79.593,-46.220,178.814,6.159,149.461
C09950=1131.922,-79.343,-46.230,178.815,6.159,149.460
C09951=1131.916,-79.093,-46.240,178.817,6.160,149.460
C09952=1131.911,-78.843,-46.249,178.820,6.160,149.459
C09953=1131.906,-78.594,-46.259,178.822,6.161,149.459
C09954=1131.900,-78.344,-46.270,178.823,6.161,149.458
C09955=1131.895,-78.094,-46.279,178.826,6.161,149.458
C09956=1131.889,-77.845,-46.289,178.828,6.162,149.457
C09957=1131.885,-77.595,-46.299,178.830,6.163,149.457
C09958=1131.878,-77.323,-46.309,178.833,6.164,149.456
C09959=1131.873,-77.052,-46.320,178.835,6.164,149.456
C09960=1131.867,-76.780,-46.331,178.838,6.165,149.455
C09961=1131.861,-76.509,-46.342,178.839,6.165,149.455
C09962=1131.856,-76.258,-46.351,178.841,6.165,149.454
C09963=1131.851,-76.009,-46.361,178.844,6.166,149.453
C09964=1131.845,-75.760,-46.371,178.846,6.167,149.453
C09965=1131.840,-75.510,-46.381,178.848,6.167,149.452
C09966=1131.834,-75.260,-46.391,178.850,6.167,149.452
C09967=1131.829,-75.010,-46.401,178.852,6.168,149.451
C09968=1131.824,-74.760,-46.411,178.854,6.169,149.451
C09969=1131.818,-74.511,-46.421,178.857,6.169,149.450
C09970=1131.813,-74.261,-46.430,178.859,6.169,149.450
C09971=1131.807,-74.011,-46.440,178.861,6.170,149.449
C09972=1131.802,-73.761,-46.451,178.863,6.171,149.449
C09973=1131.797,-73.512,-46.461,178.865,6.171,149.448
C09974=1131.792,-73.262,-46.471,178.867,6.172,149.448
C09975=1131.786,-73.012,-46.480,178.869,6.172,149.447
C09976=1131.781,-72.762,-46.491,178.872,6.173,149.447
C09977=1131.775,-72.512,-46.501,178.874,6.173,149.446
C09978=1131.771,-72.263,-46.511,178.876,6.174,149.446
C09979=1131.765,-72.014,-46.521,178.878,6.175,149.445
C09980=1131.760,-71.763,-46.532,178.880,6.175,149.445
C09981=1131.754,-71.513,-46.541,178.883,6.175,149.444
C09982=1131.749,-71.264,-46.551,178.885,6.176,149.444
C09983=1131.744,-71.015,-46.561,178.887,6.177,149.443
C09984=1131.739,-70.764,-46.571,178.889,6.177,149.443
C09985=1131.733,-70.515,-46.582,178.891,6.177,149.442
C09986=1131.727,-70.265,-46.592,178.893,6.178,149.442
C09987=1131.723,-70.016,-46.601,178.896,6.179,149.441
C09988=1131.718,-69.766,-46.612,178.898,6.179,149.440
C09989=1131.712,-69.516,-46.622,178.900,6.180,149.440
C09990=1131.706,-69.266,-46.632,178.902,6.181,149.439
C09991=1131.701,-69.016,-46.642,178.904,6.181,149.439
C09992=1131.696,-68.767,-46.652,178.906,6.182,149.438
C09993=1131.691,-68.517,-46.662,178.909,6.182,149.438
C09994=1131.685,-68.267,-46.672,178.911,6.183,149.437
C09995=1131.680,-68.017,-46.683,178.913,6.183,149.437
C09996=1131.674,-67.768,-46.693,178.915,6.183,149.436
//INST
///DATE 2021/06/25 14:32
///ATTR SC,RW,RJ
////FRAME ROBOT
///GROUP1 RB1
NOP
MOVL C00000 V=800.0 PL=0
MOVL C00001 V=800.0 PL=0
MOVL C00002 V=800.0 PL=0
MOVL C00003 V=800.0 PL=0
MOVL C00004 V=800.0 PL=0
MOVL C00005 V=800.0 PL=0
MOVL C00006 V=800.0 PL=0
MOVL C00007 V=800.0 PL=0
MOVL C00008 V=800.0 PL=0
MOVL C00009 V=800.0 PL=0
MOVL C00010 V=800.0 PL=0
MOVL C00011 V=800.0 PL=0
MOVL C00012 V=800.0 PL=0
MOVL C00013 V=800.0 PL=0
MOVL C00014 V=800.0 PL=0
MOVL C00015 V=800.0 PL=0
MOVL C00016 V=800.0 PL=0
MOVL C00017 V=800.0 PL=0
MOVL C00018 V=800.0 PL=0
MOVL C00019 V=800.0 PL=0
MOVL C00020 V=800.0 PL=0
MOVL C00021 V=800.0 PL=0
MOVL C00022 V=800.0 PL=0
MOVL C00023 V=800.0 PL=0
MOVL C00024 V=800.0 PL=0
MOVL C00025 V=800.0 PL=0
MOVL C00026 V=800.0 PL=0
MOVL C00027 V=800.0 PL=0
MOVL C00028 V=800.0 PL=0
MOVL C00029 V=800.0 PL=0
MOVL C00030 V=800.0 PL=0
MOVL C00031 V=800.0 PL=0
MOVL C00032 V=800.0 PL=0
MOVL C00033 V=800.0 PL=0
MOVL C00034 V=800.0 PL=0
MOVL C00035 V=800.0 PL=0
MOVL C00036 V=800.0 PL=0
MOVL C00037 V=800.0 PL=0
MOVL C00038 V=800.0 PL=0
MOVL C00039 V=800.0 PL=0
MOVL C00040 V=800.0 PL=0
MOVL C00041 V=800.0 PL=0
MOVL C00042 V=800.0 PL=0
MOVL C00043 V=800.0 PL=0
MOVL C00044 V=800.0 PL=0
MOVL C00045 V=800.0 PL=0
MOVL C00046 V=800.0 PL=0
MOVL C00047 V=800.0 PL=0
MOVL C00048 V=800.0 PL=0
MOVL C00049 V=800.0 PL=0
MOVL C00050 V=800.0 PL=0
MOVL C00051 V=800.0 PL=0
MOVL C00052 V=800.0 PL=0
MOVL C00053 V=800.0 PL=0
MOVL C00054 V=800.0 PL=0
MOVL C00055 V=800.0 PL=0
MOVL C00056 V=800.0 PL=0
MOVL C00057 V=800.0 PL=0
MOVL C00058 V=800.0 PL=0
MOVL C00059 V=800.0 PL=0
MOVL C00060 V=800.0 PL=0
MOVL C00061 V=800.0 PL=0
MOVL C00062 V=800.0 PL=0
MOVL C00063 V=800.0 PL=0
MOVL C00064 V=800.0 PL=0
MOVL C00065 V=800.0 PL=0
MOVL C00066 V=800.0 PL=0
MOVL C00067 V=800.0 PL=0
MOVL C00068 V=800.0 PL=0
MOVL C00069 V=800.0 PL=0
MOVL C00070 V=800.0 PL=0
MOVL C00071 V=800.0 PL=0
MOVL C00072 V=800.0 PL=0
MOVL C00073 V=800.0 PL=0
MOVL C00074 V=800.0 PL=0
MOVL C00075 V=800.0 PL=0
MOVL C00076 V=800.0 PL=0
MOVL C00077 V=800.0 PL=0
MOVL C00078 V=800.0 PL=0
MOVL C00079 V=800.0 PL=0
MOVL C00080 V=800.0 PL=0
MOVL C00081 V=800.0 PL=0
MOVL C00082 V=800.0 PL=0
MOVL C00083 V=800.0 PL=0
MOVL C00084 V=800.0 PL=0
MOVL C00085 V=800.0 PL=0
MOVL C00086 V=800.0 PL=0
MOVL C00087 V=800.0 PL=0
MOVL C00088 V=800.0 PL=0
MOVL C00089 V=800.0 PL=0
MOVL C00090 V=800.0 PL=0
MOVL C00091 V=800.0 PL=0
MOVL C00092 V=800.0 PL=0
MOVL C00093 V=800.0 PL=0
MOVL C00094 V=800.0 PL=0
MOVL C00095 V=800.0 PL=0
MOVL C00096 V=800.0 PL=0
MOVL C00097 V=800.0 PL=0
MOVL C00098 V=800.0 PL=0
MOVL C00099 V=800.0 PL=0
MOVL C00100 V=800.0 PL=0
MOVL C00101 V=800.0 PL=0
MOVL C00102 V=800.0 PL=0
MOVL C00103 V=800.0 PL=0
MOVL C00104 V=800.0 PL=0
MOVL C00105 V=800.0 PL=0
MOVL C00106 V=800.0 PL=0
MOVL C00107 V=800.0 PL=0
MOVL C00108 V=800.0 PL=0
MOVL C00109 V=800.0 PL=0
MOVL C00110 V=800.0 PL=0
MOVL C00111 V=800.0 PL=0
MOVL C00112 V=800.0 PL=0
MOVL C00113 V=800.0 PL=0
MOVL C00114 V=800.0 PL=0
MOVL C00115 V=800.0 PL=0
MOVL C00116 V=800.0 PL=0
MOVL C00117 V=800.0 PL=0
MOVL C00118 V=800.0 PL=0
MOVL C00119 V=800.0 PL=0
MOVL C00120 V=800.0 PL=0
MOVL C00121 V=800.0 PL=0
MOVL C00122 V=800.0 PL=0
MOVL C00123 V=800.0 PL=0
MOVL C00124 V=800.0 PL=0
MOVL C00125 V=800.0 PL=0
MOVL C00126 V=800.0 PL=0
MOVL C00127 V=800.0 PL=0
MOVL C00128 V=800.0 PL=0
MOVL C00129 V=800.0 PL=0
MOVL C00130 V=800.0 PL=0
MOVL C00131 V=800.0 PL=0
MOVL C00132 V=800.0 PL=0
MOVL C00133 V=800.0 PL=0
MOVL C00134 V=800.0 PL=0
MOVL C00135 V=800.0 PL=0
MOVL C00136 V=800.0 PL=0
MOVL C00137 V=800.0 PL=0
MOVL C00138 V=800.0 PL=0
MOVL C00139 V=800.0 PL=0
MOVL C00140 V=800.0 PL=0
MOVL C00141 V=800.0 PL=0
MOVL C00142 V=800.0 PL=0
MOVL C00143 V=800.0 PL=0
MOVL C00144 V=800.0 PL=0
MOVL C00145 V=800.0 PL=0
MOVL C00146 V=800.0 PL=0
MOVL C00147 V=800.0 PL=0
MOVL C00148 V=800.0 PL=0
MOVL C00149 V=800.0 PL=0
MOVL C00150 V=800.0 PL=0
MOVL C00151 V=800.0 PL=0
MOVL C00152 V=800.0 PL=0
MOVL C00153 V=800.0 PL=0
MOVL C00154 V=800.0 PL=0
MOVL C00155 V=800.0 PL=0
MOVL C00156 V=800.0 PL=0
MOVL C00157 V=800.0 PL=0
MOVL C00158 V=800.0 PL=0
MOVL C00159 V=800.0 PL=0
MOVL C00160 V=800.0 PL=0
MOVL C00161 V=800.0 PL=0
MOVL C00162 V=800.0 PL=0
MOVL C00163 V=800.0 PL=0
MOVL C00164 V=800.0 PL=0
MOVL C00165 V=800.0 PL=0
MOVL C00166 V=800.0 PL=0
MOVL C00167 V=800.0 PL=0
MOVL C00168 V=800.0 PL=0
MOVL C00169 V=800.0 PL=0
MOVL C00170 V=800.0 PL=0
MOVL C00171 V=800.0 PL=0
MOVL C00172 V=800.0 PL=0
MOVL C00173 V=800.0 PL=0
MOVL C00174 V=800.0 PL=0
MOVL C00175 V=800.0 PL=0
MOVL C00176 V=800.0 PL=0
MOVL C00177 V=800.0 PL=0
MOVL C00178 V=800.0 PL=0
MOVL C00179 V=800.0 PL=0
MOVL C00180 V=800.0 PL=0
MOVL C00181 V=800.0 PL=0
MOVL C00182 V=800.0 PL=0
MOVL C00183 V=800.0 PL=0
MOVL C00184 V=800.0 PL=0
MOVL C00185 V=800.0 PL=0
MOVL C00186 V=800.0 PL=0
MOVL C00187 V=800.0 PL=0
MOVL C00188 V=800.0 PL=0
MOVL C00189 V=800.0 PL=0
MOVL C00190 V=800.0 PL=0
MOVL C00191 V=800.0 PL=0
MOVL C00192 V=800.0 PL=0
MOVL C00193 V=800.0 PL=0
MOVL C00194 V=800.0 PL=0
MOVL C00195 V=800.0 PL=0
MOVL C00196 V=800.0 PL=0
MOVL C00197 V=800.0 PL=0
MOVL C00198 V=800.0 PL=0
MOVL C00199 V=800.0 PL=0
MOVL C00200 V=800.0 PL=0
MOVL C00201 V=800.0 PL=0
MOVL C00202 V=800.0 PL=0
MOVL C00203 V=800.0 PL=0
MOVL C00204 V=800.0 PL=0
MOVL C00205 V=800.0 PL=0
MOVL C00206 V=800.0 PL=0
MOVL C00207 V=800.0 PL=0
MOVL C00208 V=800.0 PL=0
MOVL C00209 V=800.0 PL=0
MOVL C00210 V=800.0 PL=0
MOVL C00211 V=800.0 PL=0
MOVL C00212 V=800.0 PL=0
MOVL C00213 V=800.0 PL=0
MOVL C00214 V=800.0 PL=0
MOVL C00215 V=800.0 PL=0
MOVL C00216 V=800.0 PL=0
MOVL C00217 V=800.0 PL=0
MOVL C00218 V=800.0 PL=0
MOVL C00219 V=800.0 PL=0
MOVL C00220 V=800.0 PL=0
MOVL C00221 V=800.0 PL=0
MOVL C00222 V=800.0 PL=0
MOVL C00223 V=800.0 PL=0
MOVL C00224 V=800.0 PL=0
MOVL C00225 V=800.0 PL=0
MOVL C00226 V=800.0 PL=0
MOVL C00227 V=800.0 PL=0
MOVL C00228 V=800.0 PL=0
MOVL C00229 V=800.0 PL=0
MOVL C00230 V=800.0 PL=0
MOVL C00231 V=800.0 PL=0
MOVL C00232 V=800.0 PL=0
MOVL C00233 V=800.0 PL=0
MOVL C00234 V=800.0 PL=0
MOVL C00235 V=800.0 PL=0
MOVL C00236 V=800.0 PL=0
MOVL C00237 V=800.0 PL=0
MOVL C00238 V=800.0 PL=0
MOVL C00239 V=800.0 PL=0
MOVL C00240 V=800.0 PL=0
MOVL C00241 V=800.0 PL=0
MOVL C00242 V=800.0 PL=0
MOVL C00243 V=800.0 PL=0
MOVL C00244 V=800.0 PL=0
MOVL C00245 V=800.0 PL=0
MOVL C00246 V=800.0 PL=0
MOVL C00247 V=800.0 PL=0
MOVL C00248 V=800.0 PL=0
MOVL C00249 V=800.0 PL=0
MOVL C00250 V=800.0 PL=0
MOVL C00251 V=800.0 PL=0
MOVL C00252 V=800.0 PL=0
MOVL C00253 V=800.0 PL=0
MOVL C00254 V=800.0 PL=0
MOVL C00255 V=800.0 PL=0
MOVL C00256 V=800.0 PL=0
MOVL C00257 V=800.0 PL=0
MOVL C00258 V=800.0 PL=0
MOVL C00259 V=800.0 PL=0
MOVL C00260 V=800.0 PL=0
MOVL C00261 V=800.0 PL=0
MOVL C00262 V=800.0 PL=0
MOVL C00263 V=800.0 PL=0
MOVL C00264 V=800.0 PL=0
MOVL C00265 V=800.0 PL=0
MOVL C00266 V=800.0 PL=0
MOVL C00267 V=800.0 PL=0
MOVL C00268 V=800.0 PL=0
MOVL C00269 V=800.0 PL=0
MOVL C00270 V=800.0 PL=0
MOVL C00271 V=800.0 PL=0
MOVL C00272 V=800.0 PL=0
MOVL C00273 V=800.0 PL=0
MOVL C00274 V=800.0 PL=0
MOVL C00275 V=800.0 PL=0
MOVL C00276 V=800.0 PL=0
MOVL C00277 V=800.0 PL=0
MOVL C00278 V=800.0 PL=0
MOVL C00279 V=800.0 PL=0
MOVL C00280 V=800.0 PL=0
MOVL C00281 V=800.0 PL=0
MOVL C00282 V=800.0 PL=0
MOVL C00283 V=800.0 PL=0
MOVL C00284 V=800.0 PL=0
MOVL C00285 V=800.0 PL=0
MOVL C00286 V=800.0 PL=0
MOVL C00287 V=800.0 PL=0
MOVL C00288 V=800.0 PL=0
MOVL C00289 V=800.0 PL=0
MOVL C00290 V=800.0 PL=0
MOVL C00291 V=800.0 PL=0
MOVL C00292 V=800.0 PL=0
MOVL C00293 V=800.0 PL=0
MOVL C00294 V=800.0 PL=0
MOVL C00295 V=800.0 PL=0
MOVL C00296 V=800.0 PL=0
MOVL C00297 V=800.0 PL=0
MOVL C00298 V=800.0 PL=0
MOVL C00299 V=800.0 PL=0
MOVL C00300 V=800.0 PL=0
MOVL C00301 V=800.0 PL=0
MOVL C00302 V=800.0 PL=0
MOVL C00303 V=800.0 PL=0
MOVL C00304 V=800.0 PL=0
MOVL C00305 V=800.0 PL=0
MOVL C00306 V=800.0 PL=0
MOVL C00307 V=800.0 PL=0
MOVL C00308 V=800.0 PL=0
MOVL C00309 V=800.0 PL=0
MOVL C00310 V=800.0 PL=0
MOVL C00311 V=800.0 PL=0
MOVL C00312 V=800.0 PL=0
MOVL C00313 V=800.0 PL=0
MOVL C00314 V=800.0 PL=0
MOVL C00315 V=800.0 PL=0
MOVL C00316 V=800.0 PL=0
MOVL C00317 V=800.0 PL=0
MOVL C00318 V=800.0 PL=0
MOVL C00319 V=800.0 PL=0
MOVL C00320 V=800.0 PL=0
MOVL C00321 V=800.0 PL=0
MOVL C00322 V=800.0 PL=0
MOVL C00323 V=800.0 PL=0
MOVL C00324 V=800.0 PL=0
MOVL C00325 V=800.0 PL=0
MOVL C00326 V=800.0 PL=0
MOVL C00327 V=800.0 PL=0
MOVL C00328 V=800.0 PL=0
MOVL C00329 V=800.0 PL=0
MOVL C00330 V=800.0 PL=0
MOVL C00331 V=800.0 PL=0
MOVL C00332 V=800.0 PL=0
MOVL C00333 V=800.0 PL=0
MOVL C00334 V=800.0 PL=0
MOVL C00335 V=800.0 PL=0
MOVL C00336 V=800.0 PL=0
MOVL C00337 V=800.0 PL=0
MOVL C00338 V=800.0 PL=0
MOVL C00339 V=800.0 PL=0
MOVL C00340 V=800.0 PL=0
MOVL C00341 V=800.0 PL=0
MOVL C00342 V=800.0 PL=0
MOVL C00343 V=800.0 PL=0
MOVL C00344 V=800.0 PL=0
MOVL C00345 V=800.0 PL=0
MOVL C00346 V=800.0 PL=0
MOVL C00347 V=800.0 PL=0
MOVL C00348 V=800.0 PL=0
MOVL C00349 V=800.0 PL=0
MOVL C00350 V=800.0 PL=0
MOVL C00351 V=800.0 PL=0
MOVL C00352 V=800.0 PL=0
MOVL C00353 V=800.0 PL=0
MOVL C00354 V=800.0 PL=0
MOVL C00355 V=800.0 PL=0
MOVL C00356 V=800.0 PL=0
MOVL C00357 V=800.0 PL=0
MOVL C00358 V=800.0 PL=0
MOVL C00359 V=800.0 PL=0
MOVL C00360 V=800.0 PL=0
MOVL C00361 V=800.0 PL=0
MOVL C00362 V=800.0 PL=0
MOVL C00363 V=800.0 PL=0
MOVL C00364 V=800.0 PL=0
MOVL C00365 V=800.0 PL=0
MOVL C00366 V=800.0 PL=0
MOVL C00367 V=800.0 PL=0
MOVL C00368 V=800.0 PL=0
MOVL C00369 V=800.0 PL=0
MOVL C00370 V=800.0 PL=0
MOVL C00371 V=800.0 PL=0
MOVL C00372 V=800.0 PL=0
MOVL C00373 V=800.0 PL=0
MOVL C00374 V=800.0 PL=0
MOVL C00375 V=800.0 PL=0
MOVL C00376 V=800.0 PL=0
MOVL C00377 V=800.0 PL=0
MOVL C00378 V=800.0 PL=0
MOVL C00379 V=800.0 PL=0
MOVL C00380 V=800.0 PL=0
MOVL C00381 V=800.0 PL=0
MOVL C00382 V=800.0 PL=0
MOVL C00383 V=800.0 PL=0
MOVL C00384 V=800.0 PL=0
MOVL C00385 V=800.0 PL=0
MOVL C00386 V=800.0 PL=0
MOVL C00387 V=800.0 PL=0
MOVL C00388 V=800.0 PL=0
MOVL C00389 V=800.0 PL=0
MOVL C00390 V=800.0 PL=0
MOVL C00391 V=800.0 PL=0
MOVL C00392 V=800.0 PL=0
MOVL C00393 V=800.0 PL=0
MOVL C00394 V=800.0 PL=0
MOVL C00395 V=800.0 PL=0
MOVL C00396 V=800.0 PL=0
MOVL C00397 V=800.0 PL=0
MOVL C00398 V=800.0 PL=0
MOVL C00399 V=800.0 PL=0
MOVL C00400 V=800.0 PL=0
MOVL C00401 V=800.0 PL=0
MOVL C00402 V=800.0 PL=0
MOVL C00403 V=800.0 PL=0
MOVL C00404 V=800.0 PL=0
MOVL C00405 V=800.0 PL=0
MOVL C00406 V=800.0 PL=0
MOVL C00407 V=800.0 PL=0
MOVL C00408 V=800.0 PL=0
MOVL C00409 V=800.0 PL=0
MOVL C00410 V=800.0 PL=0
MOVL C00411 V=800.0 PL=0
MOVL C00412 V=800.0 PL=0
MOVL C00413 V=800.0 PL=0
MOVL C00414 V=800.0 PL=0
MOVL C00415 V=800.0 PL=0
MOVL C00416 V=800.0 PL=0
MOVL C00417 V=800.0 PL=0
MOVL C00418 V=800.0 PL=0
MOVL C00419 V=800.0 PL=0
MOVL C00420 V=800.0 PL=0
MOVL C00421 V=800.0 PL=0
MOVL C00422 V=800.0 PL=0
MOVL C00423 V=800.0 PL=0
MOVL C00424 V=800.0 PL=0
MOVL C00425 V=800.0 PL=0
MOVL C00426 V=800.0 PL=0
MOVL C00427 V=800.0 PL=0
MOVL C00428 V=800.0 PL=0
MOVL C00429 V=800.0 PL=0
MOVL C00430 V=800.0 PL=0
MOVL C00431 V=800.0 PL=0
MOVL C00432 V=800.0 PL=0
MOVL C00433 V=800.0 PL=0
MOVL C00434 V=800.0 PL=0
MOVL C00435 V=800.0 PL=0
MOVL C00436 V=800.0 PL=0
MOVL C00437 V=800.0 PL=0
MOVL C00438 V=800.0 PL=0
MOVL C00439 V=800.0 PL=0
MOVL C00440 V=800.0 PL=0
MOVL C00441 V=800.0 PL=0
MOVL C00442 V=800.0 PL=0
MOVL C00443 V=800.0 PL=0
MOVL C00444 V=800.0 PL=0
MOVL C00445 V=800.0 PL=0
MOVL C00446 V=800.0 PL=0
MOVL C00447 V=800.0 PL=0
MOVL C00448 V=800.0 PL=0
MOVL C00449 V=800.0 PL=0
MOVL C00450 V=800.0 PL=0
MOVL C00451 V=800.0 PL=0
MOVL C00452 V=800.0 PL=0
MOVL C00453 V=800.0 PL=0
MOVL C00454 V=800.0 PL=0
MOVL C00455 V=800.0 PL=0
MOVL C00456 V=800.0 PL=0
MOVL C00457 V=800.0 PL=0
MOVL C00458 V=800.0 PL=0
MOVL C00459 V=800.0 PL=0
MOVL C00460 V=800.0 PL=0
MOVL C00461 V=800.0 PL=0
MOVL C00462 V=800.0 PL=0
MOVL C00463 V=800.0 PL=0
MOVL C00464 V=800.0 PL=0
MOVL C00465 V=800.0 PL=0
MOVL C00466 V=800.0 PL=0
MOVL C00467 V=800.0 PL=0
MOVL C00468 V=800.0 PL=0
MOVL C00469 V=800.0 PL=0
MOVL C00470 V=800.0 PL=0
MOVL C00471 V=800.0 PL=0
MOVL C00472 V=800.0 PL=0
MOVL C00473 V=800.0 PL=0
MOVL C00474 V=800.0 PL=0
MOVL C00475 V=800.0 PL=0
MOVL C00476 V=800.0 PL=0
MOVL C00477 V=800.0 PL=0
MOVL C00478 V=800.0 PL=0
MOVL C00479 V=800.0 PL=0
MOVL C00480 V=800.0 PL=0
MOVL C00481 V=800.0 PL=0
MOVL C00482 V=800.0 PL=0
MOVL C00483 V=800.0 PL=0
MOVL C00484 V=800.0 PL=0
MOVL C00485 V=800.0 PL=0
MOVL C00486 V=800.0 PL=0
MOVL C00487 V=800.0 PL=0
MOVL C00488 V=800.0 PL=0
MOVL C00489 V=800.0 PL=0
MOVL C00490 V=800.0 PL=0
MOVL C00491 V=800.0 PL=0
MOVL C00492 V=800.0 PL=0
MOVL C00493 V=800.0 PL=0
MOVL C00494 V=800.0 PL=0
MOVL C00495 V=800.0 PL=0
MOVL C00496 V=800.0 PL=0
MOVL C00497 V=800.0 PL=0
MOVL C00498 V=800.0 PL=0
MOVL C00499 V=800.0 PL=0
MOVL C00500 V=800.0 PL=0
MOVL C00501 V=800.0 PL=0
MOVL C00502 V=800.0 PL=0
MOVL C00503 V=800.0 PL=0
MOVL C00504 V=800.0 PL=0
MOVL C00505 V=800.0 PL=0
MOVL C00506 V=800.0 PL=0
MOVL C00507 V=800.0 PL=0
MOVL C00508 V=800.0 PL=0
MOVL C00509 V=800.0 PL=0
MOVL C00510 V=800.0 PL=0
MOVL C00511 V=800.0 PL=0
MOVL C00512 V=800.0 PL=0
MOVL C00513 V=800.0 PL=0
MOVL C00514 V=800.0 PL=0
MOVL C00515 V=800.0 PL=0
MOVL C00516 V=800.0 PL=0
MOVL C00517 V=800.0 PL=0
MOVL C00518 V=800.0 PL=0
MOVL C00519 V=800.0 PL=0
MOVL C00520 V=800.0 PL=0
MOVL C00521 V=800.0 PL=0
MOVL C00522 V=800.0 PL=0
MOVL C00523 V=800.0 PL=0
MOVL C00524 V=800.0 PL=0
MOVL C00525 V=800.0 PL=0
MOVL C00526 V=800.0 PL=0
MOVL C00527 V=800.0 PL=0
MOVL C00528 V=800.0 PL=0
MOVL C00529 V=800.0 PL=0
MOVL C00530 V=800.0 PL=0
MOVL C00531 V=800.0 PL=0
MOVL C00532 V=800.0 PL=0
MOVL C00533 V=800.0 PL=0
MOVL C00534 V=800.0 PL=0
MOVL C00535 V=800.0 PL=0
MOVL C00536 V=800.0 PL=0
MOVL C00537 V=800.0 PL=0
MOVL C00538 V=800.0 PL=0
MOVL C00539 V=800.0 PL=0
MOVL C00540 V=800.0 PL=0
MOVL C00541 V=800.0 PL=0
MOVL C00542 V=800.0 PL=0
MOVL C00543 V=800.0 PL=0
MOVL C00544 V=800.0 PL=0
MOVL C00545 V=800.0 PL=0
MOVL C00546 V=800.0 PL=0
MOVL C00547 V=800.0 PL=0
MOVL C00548 V=800.0 PL=0
MOVL C00549 V=800.0 PL=0
MOVL C00550 V=800.0 PL=0
MOVL C00551 V=800.0 PL=0
MOVL C00552 V=800.0 PL=0
MOVL C00553 V=800.0 PL=0
MOVL C00554 V=800.0 PL=0
MOVL C00555 V=800.0 PL=0
MOVL C00556 V=800.0 PL=0
MOVL C00557 V=800.0 PL=0
MOVL C00558 V=800.0 PL=0
MOVL C00559 V=800.0 PL=0
MOVL C00560 V=800.0 PL=0
MOVL C00561 V=800.0 PL=0
MOVL C00562 V=800.0 PL=0
MOVL C00563 V=800.0 PL=0
MOVL C00564 V=800.0 PL=0
MOVL C00565 V=800.0 PL=0
MOVL C00566 V=800.0 PL=0
MOVL C00567 V=800.0 PL=0
MOVL C00568 V=800.0 PL=0
MOVL C00569 V=800.0 PL=0
MOVL C00570 V=800.0 PL=0
MOVL C00571 V=800.0 PL=0
MOVL C00572 V=800.0 PL=0
MOVL C00573 V=800.0 PL=0
MOVL C00574 V=800.0 PL=0
MOVL C00575 V=800.0 PL=0
MOVL C00576 V=800.0 PL=0
MOVL C00577 V=800.0 PL=0
MOVL C00578 V=800.0 PL=0
MOVL C00579 V=800.0 PL=0
MOVL C00580 V=800.0 PL=0
MOVL C00581 V=800.0 PL=0
MOVL C00582 V=800.0 PL=0
MOVL C00583 V=800.0 PL=0
MOVL C00584 V=800.0 PL=0
MOVL C00585 V=800.0 PL=0
MOVL C00586 V=800.0 PL=0
MOVL C00587 V=800.0 PL=0
MOVL C00588 V=800.0 PL=0
MOVL C00589 V=800.0 PL=0
MOVL C00590 V=800.0 PL=0
MOVL C00591 V=800.0 PL=0
MOVL C00592 V=800.0 PL=0
MOVL C00593 V=800.0 PL=0
MOVL C00594 V=800.0 PL=0
MOVL C00595 V=800.0 PL=0
MOVL C00596 V=800.0 PL=0
MOVL C00597 V=800.0 PL=0
MOVL C00598 V=800.0 PL=0
MOVL C00599 V=800.0 PL=0
MOVL C00600 V=800.0 PL=0
MOVL C00601 V=800.0 PL=0
MOVL C00602 V=800.0 PL=0
MOVL C00603 V=800.0 PL=0
MOVL C00604 V=800.0 PL=0
MOVL C00605 V=800.0 PL=0
MOVL C00606 V=800.0 PL=0
MOVL C00607 V=800.0 PL=0
MOVL C00608 V=800.0 PL=0
MOVL C00609 V=800.0 PL=0
MOVL C00610 V=800.0 PL=0
MOVL C00611 V=800.0 PL=0
MOVL C00612 V=800.0 PL=0
MOVL C00613 V=800.0 PL=0
MOVL C00614 V=800.0 PL=0
MOVL C00615 V=800.0 PL=0
MOVL C00616 V=800.0 PL=0
MOVL C00617 V=800.0 PL=0
MOVL C00618 V=800.0 PL=0
MOVL C00619 V=800.0 PL=0
MOVL C00620 V=800.0 PL=0
MOVL C00621 V=800.0 PL=0
MOVL C00622 V=800.0 PL=0
MOVL C00623 V=800.0 PL=0
MOVL C00624 V=800.0 PL=0
MOVL C00625 V=800.0 PL=0
MOVL C00626 V=800.0 PL=0
MOVL C00627 V=800.0 PL=0
MOVL C00628 V=800.0 PL=0
MOVL C00629 V=800.0 PL=0
MOVL C00630 V=800.0 PL=0
MOVL C00631 V=800.0 PL=0
MOVL C00632 V=800.0 PL=0
MOVL C00633 V=800.0 PL=0
MOVL C00634 V=800.0 PL=0
MOVL C00635 V=800.0 PL=0
MOVL C00636 V=800.0 PL=0
MOVL C00637 V=800.0 PL=0
MOVL C00638 V=800.0 PL=0
MOVL C00639 V=800.0 PL=0
MOVL C00640 V=800.0 PL=0
MOVL C00641 V=800.0 PL=0
MOVL C00642 V=800.0 PL=0
MOVL C00643 V=800.0 PL=0
MOVL C00644 V=800.0 PL=0
MOVL C00645 V=800.0 PL=0
MOVL C00646 V=800.0 PL=0
MOVL C00647 V=800.0 PL=0
MOVL C00648 V=800.0 PL=0
MOVL C00649 V=800.0 PL=0
MOVL C00650 V=800.0 PL=0
MOVL C00651 V=800.0 PL=0
MOVL C00652 V=800.0 PL=0
MOVL C00653 V=800.0 PL=0
MOVL C00654 V=800.0 PL=0
MOVL C00655 V=800.0 PL=0
MOVL C00656 V=800.0 PL=0
MOVL C00657 V=800.0 PL=0
MOVL C00658 V=800.0 PL=0
MOVL C00659 V=800.0 PL=0
MOVL C00660 V=800.0 PL=0
MOVL C00661 V=800.0 PL=0
MOVL C00662 V=800.0 PL=0
MOVL C00663 V=800.0 PL=0
MOVL C00664 V=800.0 PL=0
MOVL C00665 V=800.0 PL=0
MOVL C00666 V=800.0 PL=0
MOVL C00667 V=800.0 PL=0
MOVL C00668 V=800.0 PL=0
MOVL C00669 V=800.0 PL=0
MOVL C00670 V=800.0 PL=0
MOVL C00671 V=800.0 PL=0
MOVL C00672 V=800.0 PL=0
MOVL C00673 V=800.0 PL=0
MOVL C00674 V=800.0 PL=0
MOVL C00675 V=800.0 PL=0
MOVL C00676 V=800.0 PL=0
MOVL C00677 V=800.0 PL=0
MOVL C00678 V=800.0 PL=0
MOVL C00679 V=800.0 PL=0
MOVL C00680 V=800.0 PL=0
MOVL C00681 V=800.0 PL=0
MOVL C00682 V=800.0 PL=0
MOVL C00683 V=800.0 PL=0
MOVL C00684 V=800.0 PL=0
MOVL C00685 V=800.0 PL=0
MOVL C00686 V=800.0 PL=0
MOVL C00687 V=800.0 PL=0
MOVL C00688 V=800.0 PL=0
MOVL C00689 V=800.0 PL=0
MOVL C00690 V=800.0 PL=0
MOVL C00691 V=800.0 PL=0
MOVL C00692 V=800.0 PL=0
MOVL C00693 V=800.0 PL=0
MOVL C00694 V=800.0 PL=0
MOVL C00695 V=800.0 PL=0
MOVL C00696 V=800.0 PL=0
MOVL C00697 V=800.0 PL=0
MOVL C00698 V=800.0 PL=0
MOVL C00699 V=800.0 PL=0
MOVL C00700 V=800.0 PL=0
MOVL C00701 V=800.0 PL=0
MOVL C00702 V=800.0 PL=0
MOVL C00703 V=800.0 PL=0
MOVL C00704 V=800.0 PL=0
MOVL C00705 V=800.0 PL=0
MOVL C00706 V=800.0 PL=0
MOVL C00707 V=800.0 PL=0
MOVL C00708 V=800.0 PL=0
MOVL C00709 V=800.0 PL=0
MOVL C00710 V=800.0 PL=0
MOVL C00711 V=800.0 PL=0
MOVL C00712 V=800.0 PL=0
MOVL C00713 V=800.0 PL=0
MOVL C00714 V=800.0 PL=0
MOVL C00715 V=800.0 PL=0
MOVL C00716 V=800.0 PL=0
MOVL C00717 V=800.0 PL=0
MOVL C00718 V=800.0 PL=0
MOVL C00719 V=800.0 PL=0
MOVL C00720 V=800.0 PL=0
MOVL C00721 V=800.0 PL=0
MOVL C00722 V=800.0 PL=0
MOVL C00723 V=800.0 PL=0
MOVL C00724 V=800.0 PL=0
MOVL C00725 V=800.0 PL=0
MOVL C00726 V=800.0 PL=0
MOVL C00727 V=800.0 PL=0
MOVL C00728 V=800.0 PL=0
MOVL C00729 V=800.0 PL=0
MOVL C00730 V=800.0 PL=0
MOVL C00731 V=800.0 PL=0
MOVL C00732 V=800.0 PL=0
MOVL C00733 V=800.0 PL=0
MOVL C00734 V=800.0 PL=0
MOVL C00735 V=800.0 PL=0
MOVL C00736 V=800.0 PL=0
MOVL C00737 V=800.0 PL=0
MOVL C00738 V=800.0 PL=0
MOVL C00739 V=800.0 PL=0
MOVL C00740 V=800.0 PL=0
MOVL C00741 V=800.0 PL=0
MOVL C00742 V=800.0 PL=0
MOVL C00743 V=800.0 PL=0
MOVL C00744 V=800.0 PL=0
MOVL C00745 V=800.0 PL=0
MOVL C00746 V=800.0 PL=0
MOVL C00747 V=800.0 PL=0
MOVL C00748 V=800.0 PL=0
MOVL C00749 V=800.0 PL=0
MOVL C00750 V=800.0 PL=0
MOVL C00751 V=800.0 PL=0
MOVL C00752 V=800.0 PL=0
MOVL C00753 V=800.0 PL=0
MOVL C00754 V=800.0 PL=0
MOVL C00755 V=800.0 PL=0
MOVL C00756 V=800.0 PL=0
MOVL C00757 V=800.0 PL=0
MOVL C00758 V=800.0 PL=0
MOVL C00759 V=800.0 PL=0
MOVL C00760 V=800.0 PL=0
MOVL C00761 V=800.0 PL=0
MOVL C00762 V=800.0 PL=0
MOVL C00763 V=800.0 PL=0
MOVL C00764 V=800.0 PL=0
MOVL C00765 V=800.0 PL=0
MOVL C00766 V=800.0 PL=0
MOVL C00767 V=800.0 PL=0
MOVL C00768 V=800.0 PL=0
MOVL C00769 V=800.0 PL=0
MOVL C00770 V=800.0 PL=0
MOVL C00771 V=800.0 PL=0
MOVL C00772 V=800.0 PL=0
MOVL C00773 V=800.0 PL=0
MOVL C00774 V=800.0 PL=0
MOVL C00775 V=800.0 PL=0
MOVL C00776 V=800.0 PL=0
MOVL C00777 V=800.0 PL=0
MOVL C00778 V=800.0 PL=0
MOVL C00779 V=800.0 PL=0
MOVL C00780 V=800.0 PL=0
MOVL C00781 V=800.0 PL=0
MOVL C00782 V=800.0 PL=0
MOVL C00783 V=800.0 PL=0
MOVL C00784 V=800.0 PL=0
MOVL C00785 V=800.0 PL=0
MOVL C00786 V=800.0 PL=0
MOVL C00787 V=800.0 PL=0
MOVL C00788 V=800.0 PL=0
MOVL C00789 V=800.0 PL=0
MOVL C00790 V=800.0 PL=0
MOVL C00791 V=800.0 PL=0
MOVL C00792 V=800.0 PL=0
MOVL C00793 V=800.0 PL=0
MOVL C00794 V=800.0 PL=0
MOVL C00795 V=800.0 PL=0
MOVL C00796 V=800.0 PL=0
MOVL C00797 V=800.0 PL=0
MOVL C00798 V=800.0 PL=0
MOVL C00799 V=800.0 PL=0
MOVL C00800 V=800.0 PL=0
MOVL C00801 V=800.0 PL=0
MOVL C00802 V=800.0 PL=0
MOVL C00803 V=800.0 PL=0
MOVL C00804 V=800.0 PL=0
MOVL C00805 V=800.0 PL=0
MOVL C00806 V=800.0 PL=0
MOVL C00807 V=800.0 PL=0
MOVL C00808 V=800.0 PL=0
MOVL C00809 V=800.0 PL=0
MOVL C00810 V=800.0 PL=0
MOVL C00811 V=800.0 PL=0
MOVL C00812 V=800.0 PL=0
MOVL C00813 V=800.0 PL=0
MOVL C00814 V=800.0 PL=0
MOVL C00815 V=800.0 PL=0
MOVL C00816 V=800.0 PL=0
MOVL C00817 V=800.0 PL=0
MOVL C00818 V=800.0 PL=0
MOVL C00819 V=800.0 PL=0
MOVL C00820 V=800.0 PL=0
MOVL C00821 V=800.0 PL=0
MOVL C00822 V=800.0 PL=0
MOVL C00823 V=800.0 PL=0
MOVL C00824 V=800.0 PL=0
MOVL C00825 V=800.0 PL=0
MOVL C00826 V=800.0 PL=0
MOVL C00827 V=800.0 PL=0
MOVL C00828 V=800.0 PL=0
MOVL C00829 V=800.0 PL=0
MOVL C00830 V=800.0 PL=0
MOVL C00831 V=800.0 PL=0
MOVL C00832 V=800.0 PL=0
MOVL C00833 V=800.0 PL=0
MOVL C00834 V=800.0 PL=0
MOVL C00835 V=800.0 PL=0
MOVL C00836 V=800.0 PL=0
MOVL C00837 V=800.0 PL=0
MOVL C00838 V=800.0 PL=0
MOVL C00839 V=800.0 PL=0
MOVL C00840 V=800.0 PL=0
MOVL C00841 V=800.0 PL=0
MOVL C00842 V=800.0 PL=0
MOVL C00843 V=800.0 PL=0
MOVL C00844 V=800.0 PL=0
MOVL C00845 V=800.0 PL=0
MOVL C00846 V=800.0 PL=0
MOVL C00847 V=800.0 PL=0
MOVL C00848 V=800.0 PL=0
MOVL C00849 V=800.0 PL=0
MOVL C00850 V=800.0 PL=0
MOVL C00851 V=800.0 PL=0
MOVL C00852 V=800.0 PL=0
MOVL C00853 V=800.0 PL=0
MOVL C00854 V=800.0 PL=0
MOVL C00855 V=800.0 PL=0
MOVL C00856 V=800.0 PL=0
MOVL C00857 V=800.0 PL=0
MOVL C00858 V=800.0 PL=0
MOVL C00859 V=800.0 PL=0
MOVL C00860 V=800.0 PL=0
MOVL C00861 V=800.0 PL=0
MOVL C00862 V=800.0 PL=0
MOVL C00863 V=800.0 PL=0
MOVL C00864 V=800.0 PL=0
MOVL C00865 V=800.0 PL=0
MOVL C00866 V=800.0 PL=0
MOVL C00867 V=800.0 PL=0
MOVL C00868 V=800.0 PL=0
MOVL C00869 V=800.0 PL=0
MOVL C00870 V=800.0 PL=0
MOVL C00871 V=800.0 PL=0
MOVL C00872 V=800.0 PL=0
MOVL C00873 V=800.0 PL=0
MOVL C00874 V=800.0 PL=0
MOVL C00875 V=800.0 PL=0
MOVL C00876 V=800.0 PL=0
MOVL C00877 V=800.0 PL=0
MOVL C00878 V=800.0 PL=0
MOVL C00879 V=800.0 PL=0
MOVL C00880 V=800.0 PL=0
MOVL C00881 V=800.0 PL=0
MOVL C00882 V=800.0 PL=0
MOVL C00883 V=800.0 PL=0
MOVL C00884 V=800.0 PL=0
MOVL C00885 V=800.0 PL=0
MOVL C00886 V=800.0 PL=0
MOVL C00887 V=800.0 PL=0
MOVL C00888 V=800.0 PL=0
MOVL C00889 V=800.0 PL=0
MOVL C00890 V=800.0 PL=0
MOVL C00891 V=800.0 PL=0
MOVL C00892 V=800.0 PL=0
MOVL C00893 V=800.0 PL=0
MOVL C00894 V=800.0 PL=0
MOVL C00895 V=800.0 PL=0
MOVL C00896 V=800.0 PL=0
MOVL C00897 V=800.0 PL=0
MOVL C00898 V=800.0 PL=0
MOVL C00899 V=800.0 PL=0
MOVL C00900 V=800.0 PL=0
MOVL C00901 V=800.0 PL=0
MOVL C00902 V=800.0 PL=0
MOVL C00903 V=800.0 PL=0
MOVL C00904 V=800.0 PL=0
MOVL C00905 V=800.0 PL=0
MOVL C00906 V=800.0 PL=0
MOVL C00907 V=800.0 PL=0
MOVL C00908 V=800.0 PL=0
MOVL C00909 V=800.0 PL=0
MOVL C00910 V=800.0 PL=0
MOVL C00911 V=800.0 PL=0
MOVL C00912 V=800.0 PL=0
MOVL C00913 V=800.0 PL=0
MOVL C00914 V=800.0 PL=0
MOVL C00915 V=800.0 PL=0
MOVL C00916 V=800.0 PL=0
MOVL C00917 V=800.0 PL=0
MOVL C00918 V=800.0 PL=0
MOVL C00919 V=800.0 PL=0
MOVL C00920 V=800.0 PL=0
MOVL C00921 V=800.0 PL=0
MOVL C00922 V=800.0 PL=0
MOVL C00923 V=800.0 PL=0
MOVL C00924 V=800.0 PL=0
MOVL C00925 V=800.0 PL=0
MOVL C00926 V=800.0 PL=0
MOVL C00927 V=800.0 PL=0
MOVL C00928 V=800.0 PL=0
MOVL C00929 V=800.0 PL=0
MOVL C00930 V=800.0 PL=0
MOVL C00931 V=800.0 PL=0
MOVL C00932 V=800.0 PL=0
MOVL C00933 V=800.0 PL=0
MOVL C00934 V=800.0 PL=0
MOVL C00935 V=800.0 PL=0
MOVL C00936 V=800.0 PL=0
MOVL C00937 V=800.0 PL=0
MOVL C00938 V=800.0 PL=0
MOVL C00939 V=800.0 PL=0
MOVL C00940 V=800.0 PL=0
MOVL C00941 V=800.0 PL=0
MOVL C00942 V=800.0 PL=0
MOVL C00943 V=800.0 PL=0
MOVL C00944 V=800.0 PL=0
MOVL C00945 V=800.0 PL=0
MOVL C00946 V=800.0 PL=0
MOVL C00947 V=800.0 PL=0
MOVL C00948 V=800.0 PL=0
MOVL C00949 V=800.0 PL=0
MOVL C00950 V=800.0 PL=0
MOVL C00951 V=800.0 PL=0
MOVL C00952 V=800.0 PL=0
MOVL C00953 V=800.0 PL=0
MOVL C00954 V=800.0 PL=0
MOVL C00955 V=800.0 PL=0
MOVL C00956 V=800.0 PL=0
MOVL C00957 V=800.0 PL=0
MOVL C00958 V=800.0 PL=0
MOVL C00959 V=800.0 PL=0
MOVL C00960 V=800.0 PL=0
MOVL C00961 V=800.0 PL=0
MOVL C00962 V=800.0 PL=0
MOVL C00963 V=800.0 PL=0
MOVL C00964 V=800.0 PL=0
MOVL C00965 V=800.0 PL=0
MOVL C00966 V=800.0 PL=0
MOVL C00967 V=800.0 PL=0
MOVL C00968 V=800.0 PL=0
MOVL C00969 V=800.0 PL=0
MOVL C00970 V=800.0 PL=0
MOVL C00971 V=800.0 PL=0
MOVL C00972 V=800.0 PL=0
MOVL C00973 V=800.0 PL=0
MOVL C00974 V=800.0 PL=0
MOVL C00975 V=800.0 PL=0
MOVL C00976 V=800.0 PL=0
MOVL C00977 V=800.0 PL=0
MOVL C00978 V=800.0 PL=0
MOVL C00979 V=800.0 PL=0
MOVL C00980 V=800.0 PL=0
MOVL C00981 V=800.0 PL=0
MOVL C00982 V=800.0 PL=0
MOVL C00983 V=800.0 PL=0
MOVL C00984 V=800.0 PL=0
MOVL C00985 V=800.0 PL=0
MOVL C00986 V=800.0 PL=0
MOVL C00987 V=800.0 PL=0
MOVL C00988 V=800.0 PL=0
MOVL C00989 V=800.0 PL=0
MOVL C00990 V=800.0 PL=0
MOVL C00991 V=800.0 PL=0
MOVL C00992 V=800.0 PL=0
MOVL C00993 V=800.0 PL=0
MOVL C00994 V=800.0 PL=0
MOVL C00995 V=800.0 PL=0
MOVL C00996 V=800.0 PL=0
MOVL C00997 V=800.0 PL=0
MOVL C00998 V=800.0 PL=0
MOVL C00999 V=800.0 PL=0
MOVL C01000 V=800.0 PL=0
MOVL C01001 V=800.0 PL=0
MOVL C01002 V=800.0 PL=0
MOVL C01003 V=800.0 PL=0
MOVL C01004 V=800.0 PL=0
MOVL C01005 V=800.0 PL=0
MOVL C01006 V=800.0 PL=0
MOVL C01007 V=800.0 PL=0
MOVL C01008 V=800.0 PL=0
MOVL C01009 V=800.0 PL=0
MOVL C01010 V=800.0 PL=0
MOVL C01011 V=800.0 PL=0
MOVL C01012 V=800.0 PL=0
MOVL C01013 V=800.0 PL=0
MOVL C01014 V=800.0 PL=0
MOVL C01015 V=800.0 PL=0
MOVL C01016 V=800.0 PL=0
MOVL C01017 V=800.0 PL=0
MOVL C01018 V=800.0 PL=0
MOVL C01019 V=800.0 PL=0
MOVL C01020 V=800.0 PL=0
MOVL C01021 V=800.0 PL=0
MOVL C01022 V=800.0 PL=0
MOVL C01023 V=800.0 PL=0
MOVL C01024 V=800.0 PL=0
MOVL C01025 V=800.0 PL=0
MOVL C01026 V=800.0 PL=0
MOVL C01027 V=800.0 PL=0
MOVL C01028 V=800.0 PL=0
MOVL C01029 V=800.0 PL=0
MOVL C01030 V=800.0 PL=0
MOVL C01031 V=800.0 PL=0
MOVL C01032 V=800.0 PL=0
MOVL C01033 V=800.0 PL=0
MOVL C01034 V=800.0 PL=0
MOVL C01035 V=800.0 PL=0
MOVL C01036 V=800.0 PL=0
MOVL C01037 V=800.0 PL=0
MOVL C01038 V=800.0 PL=0
MOVL C01039 V=800.0 PL=0
MOVL C01040 V=800.0 PL=0
MOVL C01041 V=800.0 PL=0
MOVL C01042 V=800.0 PL=0
MOVL C01043 V=800.0 PL=0
MOVL C01044 V=800.0 PL=0
MOVL C01045 V=800.0 PL=0
MOVL C01046 V=800.0 PL=0
MOVL C01047 V=800.0 PL=0
MOVL C01048 V=800.0 PL=0
MOVL C01049 V=800.0 PL=0
MOVL C01050 V=800.0 PL=0
MOVL C01051 V=800.0 PL=0
MOVL C01052 V=800.0 PL=0
MOVL C01053 V=800.0 PL=0
MOVL C01054 V=800.0 PL=0
MOVL C01055 V=800.0 PL=0
MOVL C01056 V=800.0 PL=0
MOVL C01057 V=800.0 PL=0
MOVL C01058 V=800.0 PL=0
MOVL C01059 V=800.0 PL=0
MOVL C01060 V=800.0 PL=0
MOVL C01061 V=800.0 PL=0
MOVL C01062 V=800.0 PL=0
MOVL C01063 V=800.0 PL=0
MOVL C01064 V=800.0 PL=0
MOVL C01065 V=800.0 PL=0
MOVL C01066 V=800.0 PL=0
MOVL C01067 V=800.0 PL=0
MOVL C01068 V=800.0 PL=0
MOVL C01069 V=800.0 PL=0
MOVL C01070 V=800.0 PL=0
MOVL C01071 V=800.0 PL=0
MOVL C01072 V=800.0 PL=0
MOVL C01073 V=800.0 PL=0
MOVL C01074 V=800.0 PL=0
MOVL C01075 V=800.0 PL=0
MOVL C01076 V=800.0 PL=0
MOVL C01077 V=800.0 PL=0
MOVL C01078 V=800.0 PL=0
MOVL C01079 V=800.0 PL=0
MOVL C01080 V=800.0 PL=0
MOVL C01081 V=800.0 PL=0
MOVL C01082 V=800.0 PL=0
MOVL C01083 V=800.0 PL=0
MOVL C01084 V=800.0 PL=0
MOVL C01085 V=800.0 PL=0
MOVL C01086 V=800.0 PL=0
MOVL C01087 V=800.0 PL=0
MOVL C01088 V=800.0 PL=0
MOVL C01089 V=800.0 PL=0
MOVL C01090 V=800.0 PL=0
MOVL C01091 V=800.0 PL=0
MOVL C01092 V=800.0 PL=0
MOVL C01093 V=800.0 PL=0
MOVL C01094 V=800.0 PL=0
MOVL C01095 V=800.0 PL=0
MOVL C01096 V=800.0 PL=0
MOVL C01097 V=800.0 PL=0
MOVL C01098 V=800.0 PL=0
MOVL C01099 V=800.0 PL=0
MOVL C01100 V=800.0 PL=0
MOVL C01101 V=800.0 PL=0
MOVL C01102 V=800.0 PL=0
MOVL C01103 V=800.0 PL=0
MOVL C01104 V=800.0 PL=0
MOVL C01105 V=800.0 PL=0
MOVL C01106 V=800.0 PL=0
MOVL C01107 V=800.0 PL=0
MOVL C01108 V=800.0 PL=0
MOVL C01109 V=800.0 PL=0
MOVL C01110 V=800.0 PL=0
MOVL C01111 V=800.0 PL=0
MOVL C01112 V=800.0 PL=0
MOVL C01113 V=800.0 PL=0
MOVL C01114 V=800.0 PL=0
MOVL C01115 V=800.0 PL=0
MOVL C01116 V=800.0 PL=0
MOVL C01117 V=800.0 PL=0
MOVL C01118 V=800.0 PL=0
MOVL C01119 V=800.0 PL=0
MOVL C01120 V=800.0 PL=0
MOVL C01121 V=800.0 PL=0
MOVL C01122 V=800.0 PL=0
MOVL C01123 V=800.0 PL=0
MOVL C01124 V=800.0 PL=0
MOVL C01125 V=800.0 PL=0
MOVL C01126 V=800.0 PL=0
MOVL C01127 V=800.0 PL=0
MOVL C01128 V=800.0 PL=0
MOVL C01129 V=800.0 PL=0
MOVL C01130 V=800.0 PL=0
MOVL C01131 V=800.0 PL=0
MOVL C01132 V=800.0 PL=0
MOVL C01133 V=800.0 PL=0
MOVL C01134 V=800.0 PL=0
MOVL C01135 V=800.0 PL=0
MOVL C01136 V=800.0 PL=0
MOVL C01137 V=800.0 PL=0
MOVL C01138 V=800.0 PL=0
MOVL C01139 V=800.0 PL=0
MOVL C01140 V=800.0 PL=0
MOVL C01141 V=800.0 PL=0
MOVL C01142 V=800.0 PL=0
MOVL C01143 V=800.0 PL=0
MOVL C01144 V=800.0 PL=0
MOVL C01145 V=800.0 PL=0
MOVL C01146 V=800.0 PL=0
MOVL C01147 V=800.0 PL=0
MOVL C01148 V=800.0 PL=0
MOVL C01149 V=800.0 PL=0
MOVL C01150 V=800.0 PL=0
MOVL C01151 V=800.0 PL=0
MOVL C01152 V=800.0 PL=0
MOVL C01153 V=800.0 PL=0
MOVL C01154 V=800.0 PL=0
MOVL C01155 V=800.0 PL=0
MOVL C01156 V=800.0 PL=0
MOVL C01157 V=800.0 PL=0
MOVL C01158 V=800.0 PL=0
MOVL C01159 V=800.0 PL=0
MOVL C01160 V=800.0 PL=0
MOVL C01161 V=800.0 PL=0
MOVL C01162 V=800.0 PL=0
MOVL C01163 V=800.0 PL=0
MOVL C01164 V=800.0 PL=0
MOVL C01165 V=800.0 PL=0
MOVL C01166 V=800.0 PL=0
MOVL C01167 V=800.0 PL=0
MOVL C01168 V=800.0 PL=0
MOVL C01169 V=800.0 PL=0
MOVL C01170 V=800.0 PL=0
MOVL C01171 V=800.0 PL=0
MOVL C01172 V=800.0 PL=0
MOVL C01173 V=800.0 PL=0
MOVL C01174 V=800.0 PL=0
MOVL C01175 V=800.0 PL=0
MOVL C01176 V=800.0 PL=0
MOVL C01177 V=800.0 PL=0
MOVL C01178 V=800.0 PL=0
MOVL C01179 V=800.0 PL=0
MOVL C01180 V=800.0 PL=0
MOVL C01181 V=800.0 PL=0
MOVL C01182 V=800.0 PL=0
MOVL C01183 V=800.0 PL=0
MOVL C01184 V=800.0 PL=0
MOVL C01185 V=800.0 PL=0
MOVL C01186 V=800.0 PL=0
MOVL C01187 V=800.0 PL=0
MOVL C01188 V=800.0 PL=0
MOVL C01189 V=800.0 PL=0
MOVL C01190 V=800.0 PL=0
MOVL C01191 V=800.0 PL=0
MOVL C01192 V=800.0 PL=0
MOVL C01193 V=800.0 PL=0
MOVL C01194 V=800.0 PL=0
MOVL C01195 V=800.0 PL=0
MOVL C01196 V=800.0 PL=0
MOVL C01197 V=800.0 PL=0
MOVL C01198 V=800.0 PL=0
MOVL C01199 V=800.0 PL=0
MOVL C01200 V=800.0 PL=0
MOVL C01201 V=800.0 PL=0
MOVL C01202 V=800.0 PL=0
MOVL C01203 V=800.0 PL=0
MOVL C01204 V=800.0 PL=0
MOVL C01205 V=800.0 PL=0
MOVL C01206 V=800.0 PL=0
MOVL C01207 V=800.0 PL=0
MOVL C01208 V=800.0 PL=0
MOVL C01209 V=800.0 PL=0
MOVL C01210 V=800.0 PL=0
MOVL C01211 V=800.0 PL=0
MOVL C01212 V=800.0 PL=0
MOVL C01213 V=800.0 PL=0
MOVL C01214 V=800.0 PL=0
MOVL C01215 V=800.0 PL=0
MOVL C01216 V=800.0 PL=0
MOVL C01217 V=800.0 PL=0
MOVL C01218 V=800.0 PL=0
MOVL C01219 V=800.0 PL=0
MOVL C01220 V=800.0 PL=0
MOVL C01221 V=800.0 PL=0
MOVL C01222 V=800.0 PL=0
MOVL C01223 V=800.0 PL=0
MOVL C01224 V=800.0 PL=0
MOVL C01225 V=800.0 PL=0
MOVL C01226 V=800.0 PL=0
MOVL C01227 V=800.0 PL=0
MOVL C01228 V=800.0 PL=0
MOVL C01229 V=800.0 PL=0
MOVL C01230 V=800.0 PL=0
MOVL C01231 V=800.0 PL=0
MOVL C01232 V=800.0 PL=0
MOVL C01233 V=800.0 PL=0
MOVL C01234 V=800.0 PL=0
MOVL C01235 V=800.0 PL=0
MOVL C01236 V=800.0 PL=0
MOVL C01237 V=800.0 PL=0
MOVL C01238 V=800.0 PL=0
MOVL C01239 V=800.0 PL=0
MOVL C01240 V=800.0 PL=0
MOVL C01241 V=800.0 PL=0
MOVL C01242 V=800.0 PL=0
MOVL C01243 V=800.0 PL=0
MOVL C01244 V=800.0 PL=0
MOVL C01245 V=800.0 PL=0
MOVL C01246 V=800.0 PL=0
MOVL C01247 V=800.0 PL=0
MOVL C01248 V=800.0 PL=0
MOVL C01249 V=800.0 PL=0
MOVL C01250 V=800.0 PL=0
MOVL C01251 V=800.0 PL=0
MOVL C01252 V=800.0 PL=0
MOVL C01253 V=800.0 PL=0
MOVL C01254 V=800.0 PL=0
MOVL C01255 V=800.0 PL=0
MOVL C01256 V=800.0 PL=0
MOVL C01257 V=800.0 PL=0
MOVL C01258 V=800.0 PL=0
MOVL C01259 V=800.0 PL=0
MOVL C01260 V=800.0 PL=0
MOVL C01261 V=800.0 PL=0
MOVL C01262 V=800.0 PL=0
MOVL C01263 V=800.0 PL=0
MOVL C01264 V=800.0 PL=0
MOVL C01265 V=800.0 PL=0
MOVL C01266 V=800.0 PL=0
MOVL C01267 V=800.0 PL=0
MOVL C01268 V=800.0 PL=0
MOVL C01269 V=800.0 PL=0
MOVL C01270 V=800.0 PL=0
MOVL C01271 V=800.0 PL=0
MOVL C01272 V=800.0 PL=0
MOVL C01273 V=800.0 PL=0
MOVL C01274 V=800.0 PL=0
MOVL C01275 V=800.0 PL=0
MOVL C01276 V=800.0 PL=0
MOVL C01277 V=800.0 PL=0
MOVL C01278 V=800.0 PL=0
MOVL C01279 V=800.0 PL=0
MOVL C01280 V=800.0 PL=0
MOVL C01281 V=800.0 PL=0
MOVL C01282 V=800.0 PL=0
MOVL C01283 V=800.0 PL=0
MOVL C01284 V=800.0 PL=0
MOVL C01285 V=800.0 PL=0
MOVL C01286 V=800.0 PL=0
MOVL C01287 V=800.0 PL=0
MOVL C01288 V=800.0 PL=0
MOVL C01289 V=800.0 PL=0
MOVL C01290 V=800.0 PL=0
MOVL C01291 V=800.0 PL=0
MOVL C01292 V=800.0 PL=0
MOVL C01293 V=800.0 PL=0
MOVL C01294 V=800.0 PL=0
MOVL C01295 V=800.0 PL=0
MOVL C01296 V=800.0 PL=0
MOVL C01297 V=800.0 PL=0
MOVL C01298 V=800.0 PL=0
MOVL C01299 V=800.0 PL=0
MOVL C01300 V=800.0 PL=0
MOVL C01301 V=800.0 PL=0
MOVL C01302 V=800.0 PL=0
MOVL C01303 V=800.0 PL=0
MOVL C01304 V=800.0 PL=0
MOVL C01305 V=800.0 PL=0
MOVL C01306 V=800.0 PL=0
MOVL C01307 V=800.0 PL=0
MOVL C01308 V=800.0 PL=0
MOVL C01309 V=800.0 PL=0
MOVL C01310 V=800.0 PL=0
MOVL C01311 V=800.0 PL=0
MOVL C01312 V=800.0 PL=0
MOVL C01313 V=800.0 PL=0
MOVL C01314 V=800.0 PL=0
MOVL C01315 V=800.0 PL=0
MOVL C01316 V=800.0 PL=0
MOVL C01317 V=800.0 PL=0
MOVL C01318 V=800.0 PL=0
MOVL C01319 V=800.0 PL=0
MOVL C01320 V=800.0 PL=0
MOVL C01321 V=800.0 PL=0
MOVL C01322 V=800.0 PL=0
MOVL C01323 V=800.0 PL=0
MOVL C01324 V=800.0 PL=0
MOVL C01325 V=800.0 PL=0
MOVL C01326 V=800.0 PL=0
MOVL C01327 V=800.0 PL=0
MOVL C01328 V=800.0 PL=0
MOVL C01329 V=800.0 PL=0
MOVL C01330 V=800.0 PL=0
MOVL C01331 V=800.0 PL=0
MOVL C01332 V=800.0 PL=0
MOVL C01333 V=800.0 PL=0
MOVL C01334 V=800.0 PL=0
MOVL C01335 V=800.0 PL=0
MOVL C01336 V=800.0 PL=0
MOVL C01337 V=800.0 PL=0
MOVL C01338 V=800.0 PL=0
MOVL C01339 V=800.0 PL=0
MOVL C01340 V=800.0 PL=0
MOVL C01341 V=800.0 PL=0
MOVL C01342 V=800.0 PL=0
MOVL C01343 V=800.0 PL=0
MOVL C01344 V=800.0 PL=0
MOVL C01345 V=800.0 PL=0
MOVL C01346 V=800.0 PL=0
MOVL C01347 V=800.0 PL=0
MOVL C01348 V=800.0 PL=0
MOVL C01349 V=800.0 PL=0
MOVL C01350 V=800.0 PL=0
MOVL C01351 V=800.0 PL=0
MOVL C01352 V=800.0 PL=0
MOVL C01353 V=800.0 PL=0
MOVL C01354 V=800.0 PL=0
MOVL C01355 V=800.0 PL=0
MOVL C01356 V=800.0 PL=0
MOVL C01357 V=800.0 PL=0
MOVL C01358 V=800.0 PL=0
MOVL C01359 V=800.0 PL=0
MOVL C01360 V=800.0 PL=0
MOVL C01361 V=800.0 PL=0
MOVL C01362 V=800.0 PL=0
MOVL C01363 V=800.0 PL=0
MOVL C01364 V=800.0 PL=0
MOVL C01365 V=800.0 PL=0
MOVL C01366 V=800.0 PL=0
MOVL C01367 V=800.0 PL=0
MOVL C01368 V=800.0 PL=0
MOVL C01369 V=800.0 PL=0
MOVL C01370 V=800.0 PL=0
MOVL C01371 V=800.0 PL=0
MOVL C01372 V=800.0 PL=0
MOVL C01373 V=800.0 PL=0
MOVL C01374 V=800.0 PL=0
MOVL C01375 V=800.0 PL=0
MOVL C01376 V=800.0 PL=0
MOVL C01377 V=800.0 PL=0
MOVL C01378 V=800.0 PL=0
MOVL C01379 V=800.0 PL=0
MOVL C01380 V=800.0 PL=0
MOVL C01381 V=800.0 PL=0
MOVL C01382 V=800.0 PL=0
MOVL C01383 V=800.0 PL=0
MOVL C01384 V=800.0 PL=0
MOVL C01385 V=800.0 PL=0
MOVL C01386 V=800.0 PL=0
MOVL C01387 V=800.0 PL=0
MOVL C01388 V=800.0 PL=0
MOVL C01389 V=800.0 PL=0
MOVL C01390 V=800.0 PL=0
MOVL C01391 V=800.0 PL=0
MOVL C01392 V=800.0 PL=0
MOVL C01393 V=800.0 PL=0
MOVL C01394 V=800.0 PL=0
MOVL C01395 V=800.0 PL=0
MOVL C01396 V=800.0 PL=0
MOVL C01397 V=800.0 PL=0
MOVL C01398 V=800.0 PL=0
MOVL C01399 V=800.0 PL=0
MOVL C01400 V=800.0 PL=0
MOVL C01401 V=800.0 PL=0
MOVL C01402 V=800.0 PL=0
MOVL C01403 V=800.0 PL=0
MOVL C01404 V=800.0 PL=0
MOVL C01405 V=800.0 PL=0
MOVL C01406 V=800.0 PL=0
MOVL C01407 V=800.0 PL=0
MOVL C01408 V=800.0 PL=0
MOVL C01409 V=800.0 PL=0
MOVL C01410 V=800.0 PL=0
MOVL C01411 V=800.0 PL=0
MOVL C01412 V=800.0 PL=0
MOVL C01413 V=800.0 PL=0
MOVL C01414 V=800.0 PL=0
MOVL C01415 V=800.0 PL=0
MOVL C01416 V=800.0 PL=0
MOVL C01417 V=800.0 PL=0
MOVL C01418 V=800.0 PL=0
MOVL C01419 V=800.0 PL=0
MOVL C01420 V=800.0 PL=0
MOVL C01421 V=800.0 PL=0
MOVL C01422 V=800.0 PL=0
MOVL C01423 V=800.0 PL=0
MOVL C01424 V=800.0 PL=0
MOVL C01425 V=800.0 PL=0
MOVL C01426 V=800.0 PL=0
MOVL C01427 V=800.0 PL=0
MOVL C01428 V=800.0 PL=0
MOVL C01429 V=800.0 PL=0
MOVL C01430 V=800.0 PL=0
MOVL C01431 V=800.0 PL=0
MOVL C01432 V=800.0 PL=0
MOVL C01433 V=800.0 PL=0
MOVL C01434 V=800.0 PL=0
MOVL C01435 V=800.0 PL=0
MOVL C01436 V=800.0 PL=0
MOVL C01437 V=800.0 PL=0
MOVL C01438 V=800.0 PL=0
MOVL C01439 V=800.0 PL=0
MOVL C01440 V=800.0 PL=0
MOVL C01441 V=800.0 PL=0
MOVL C01442 V=800.0 PL=0
MOVL C01443 V=800.0 PL=0
MOVL C01444 V=800.0 PL=0
MOVL C01445 V=800.0 PL=0
MOVL C01446 V=800.0 PL=0
MOVL C01447 V=800.0 PL=0
MOVL C01448 V=800.0 PL=0
MOVL C01449 V=800.0 PL=0
MOVL C01450 V=800.0 PL=0
MOVL C01451 V=800.0 PL=0
MOVL C01452 V=800.0 PL=0
MOVL C01453 V=800.0 PL=0
MOVL C01454 V=800.0 PL=0
MOVL C01455 V=800.0 PL=0
MOVL C01456 V=800.0 PL=0
MOVL C01457 V=800.0 PL=0
MOVL C01458 V=800.0 PL=0
MOVL C01459 V=800.0 PL=0
MOVL C01460 V=800.0 PL=0
MOVL C01461 V=800.0 PL=0
MOVL C01462 V=800.0 PL=0
MOVL C01463 V=800.0 PL=0
MOVL C01464 V=800.0 PL=0
MOVL C01465 V=800.0 PL=0
MOVL C01466 V=800.0 PL=0
MOVL C01467 V=800.0 PL=0
MOVL C01468 V=800.0 PL=0
MOVL C01469 V=800.0 PL=0
MOVL C01470 V=800.0 PL=0
MOVL C01471 V=800.0 PL=0
MOVL C01472 V=800.0 PL=0
MOVL C01473 V=800.0 PL=0
MOVL C01474 V=800.0 PL=0
MOVL C01475 V=800.0 PL=0
MOVL C01476 V=800.0 PL=0
MOVL C01477 V=800.0 PL=0
MOVL C01478 V=800.0 PL=0
MOVL C01479 V=800.0 PL=0
MOVL C01480 V=800.0 PL=0
MOVL C01481 V=800.0 PL=0
MOVL C01482 V=800.0 PL=0
MOVL C01483 V=800.0 PL=0
MOVL C01484 V=800.0 PL=0
MOVL C01485 V=800.0 PL=0
MOVL C01486 V=800.0 PL=0
MOVL C01487 V=800.0 PL=0
MOVL C01488 V=800.0 PL=0
MOVL C01489 V=800.0 PL=0
MOVL C01490 V=800.0 PL=0
MOVL C01491 V=800.0 PL=0
MOVL C01492 V=800.0 PL=0
MOVL C01493 V=800.0 PL=0
MOVL C01494 V=800.0 PL=0
MOVL C01495 V=800.0 PL=0
MOVL C01496 V=800.0 PL=0
MOVL C01497 V=800.0 PL=0
MOVL C01498 V=800.0 PL=0
MOVL C01499 V=800.0 PL=0
MOVL C01500 V=800.0 PL=0
MOVL C01501 V=800.0 PL=0
MOVL C01502 V=800.0 PL=0
MOVL C01503 V=800.0 PL=0
MOVL C01504 V=800.0 PL=0
MOVL C01505 V=800.0 PL=0
MOVL C01506 V=800.0 PL=0
MOVL C01507 V=800.0 PL=0
MOVL C01508 V=800.0 PL=0
MOVL C01509 V=800.0 PL=0
MOVL C01510 V=800.0 PL=0
MOVL C01511 V=800.0 PL=0
MOVL C01512 V=800.0 PL=0
MOVL C01513 V=800.0 PL=0
MOVL C01514 V=800.0 PL=0
MOVL C01515 V=800.0 PL=0
MOVL C01516 V=800.0 PL=0
MOVL C01517 V=800.0 PL=0
MOVL C01518 V=800.0 PL=0
MOVL C01519 V=800.0 PL=0
MOVL C01520 V=800.0 PL=0
MOVL C01521 V=800.0 PL=0
MOVL C01522 V=800.0 PL=0
MOVL C01523 V=800.0 PL=0
MOVL C01524 V=800.0 PL=0
MOVL C01525 V=800.0 PL=0
MOVL C01526 V=800.0 PL=0
MOVL C01527 V=800.0 PL=0
MOVL C01528 V=800.0 PL=0
MOVL C01529 V=800.0 PL=0
MOVL C01530 V=800.0 PL=0
MOVL C01531 V=800.0 PL=0
MOVL C01532 V=800.0 PL=0
MOVL C01533 V=800.0 PL=0
MOVL C01534 V=800.0 PL=0
MOVL C01535 V=800.0 PL=0
MOVL C01536 V=800.0 PL=0
MOVL C01537 V=800.0 PL=0
MOVL C01538 V=800.0 PL=0
MOVL C01539 V=800.0 PL=0
MOVL C01540 V=800.0 PL=0
MOVL C01541 V=800.0 PL=0
MOVL C01542 V=800.0 PL=0
MOVL C01543 V=800.0 PL=0
MOVL C01544 V=800.0 PL=0
MOVL C01545 V=800.0 PL=0
MOVL C01546 V=800.0 PL=0
MOVL C01547 V=800.0 PL=0
MOVL C01548 V=800.0 PL=0
MOVL C01549 V=800.0 PL=0
MOVL C01550 V=800.0 PL=0
MOVL C01551 V=800.0 PL=0
MOVL C01552 V=800.0 PL=0
MOVL C01553 V=800.0 PL=0
MOVL C01554 V=800.0 PL=0
MOVL C01555 V=800.0 PL=0
MOVL C01556 V=800.0 PL=0
MOVL C01557 V=800.0 PL=0
MOVL C01558 V=800.0 PL=0
MOVL C01559 V=800.0 PL=0
MOVL C01560 V=800.0 PL=0
MOVL C01561 V=800.0 PL=0
MOVL C01562 V=800.0 PL=0
MOVL C01563 V=800.0 PL=0
MOVL C01564 V=800.0 PL=0
MOVL C01565 V=800.0 PL=0
MOVL C01566 V=800.0 PL=0
MOVL C01567 V=800.0 PL=0
MOVL C01568 V=800.0 PL=0
MOVL C01569 V=800.0 PL=0
MOVL C01570 V=800.0 PL=0
MOVL C01571 V=800.0 PL=0
MOVL C01572 V=800.0 PL=0
MOVL C01573 V=800.0 PL=0
MOVL C01574 V=800.0 PL=0
MOVL C01575 V=800.0 PL=0
MOVL C01576 V=800.0 PL=0
MOVL C01577 V=800.0 PL=0
MOVL C01578 V=800.0 PL=0
MOVL C01579 V=800.0 PL=0
MOVL C01580 V=800.0 PL=0
MOVL C01581 V=800.0 PL=0
MOVL C01582 V=800.0 PL=0
MOVL C01583 V=800.0 PL=0
MOVL C01584 V=800.0 PL=0
MOVL C01585 V=800.0 PL=0
MOVL C01586 V=800.0 PL=0
MOVL C01587 V=800.0 PL=0
MOVL C01588 V=800.0 PL=0
MOVL C01589 V=800.0 PL=0
MOVL C01590 V=800.0 PL=0
MOVL C01591 V=800.0 PL=0
MOVL C01592 V=800.0 PL=0
MOVL C01593 V=800.0 PL=0
MOVL C01594 V=800.0 PL=0
MOVL C01595 V=800.0 PL=0
MOVL C01596 V=800.0 PL=0
MOVL C01597 V=800.0 PL=0
MOVL C01598 V=800.0 PL=0
MOVL C01599 V=800.0 PL=0
MOVL C01600 V=800.0 PL=0
MOVL C01601 V=800.0 PL=0
MOVL C01602 V=800.0 PL=0
MOVL C01603 V=800.0 PL=0
MOVL C01604 V=800.0 PL=0
MOVL C01605 V=800.0 PL=0
MOVL C01606 V=800.0 PL=0
MOVL C01607 V=800.0 PL=0
MOVL C01608 V=800.0 PL=0
MOVL C01609 V=800.0 PL=0
MOVL C01610 V=800.0 PL=0
MOVL C01611 V=800.0 PL=0
MOVL C01612 V=800.0 PL=0
MOVL C01613 V=800.0 PL=0
MOVL C01614 V=800.0 PL=0
MOVL C01615 V=800.0 PL=0
MOVL C01616 V=800.0 PL=0
MOVL C01617 V=800.0 PL=0
MOVL C01618 V=800.0 PL=0
MOVL C01619 V=800.0 PL=0
MOVL C01620 V=800.0 PL=0
MOVL C01621 V=800.0 PL=0
MOVL C01622 V=800.0 PL=0
MOVL C01623 V=800.0 PL=0
MOVL C01624 V=800.0 PL=0
MOVL C01625 V=800.0 PL=0
MOVL C01626 V=800.0 PL=0
MOVL C01627 V=800.0 PL=0
MOVL C01628 V=800.0 PL=0
MOVL C01629 V=800.0 PL=0
MOVL C01630 V=800.0 PL=0
MOVL C01631 V=800.0 PL=0
MOVL C01632 V=800.0 PL=0
MOVL C01633 V=800.0 PL=0
MOVL C01634 V=800.0 PL=0
MOVL C01635 V=800.0 PL=0
MOVL C01636 V=800.0 PL=0
MOVL C01637 V=800.0 PL=0
MOVL C01638 V=800.0 PL=0
MOVL C01639 V=800.0 PL=0
MOVL C01640 V=800.0 PL=0
MOVL C01641 V=800.0 PL=0
MOVL C01642 V=800.0 PL=0
MOVL C01643 V=800.0 PL=0
MOVL C01644 V=800.0 PL=0
MOVL C01645 V=800.0 PL=0
MOVL C01646 V=800.0 PL=0
MOVL C01647 V=800.0 PL=0
MOVL C01648 V=800.0 PL=0
MOVL C01649 V=800.0 PL=0
MOVL C01650 V=800.0 PL=0
MOVL C01651 V=800.0 PL=0
MOVL C01652 V=800.0 PL=0
MOVL C01653 V=800.0 PL=0
MOVL C01654 V=800.0 PL=0
MOVL C01655 V=800.0 PL=0
MOVL C01656 V=800.0 PL=0
MOVL C01657 V=800.0 PL=0
MOVL C01658 V=800.0 PL=0
MOVL C01659 V=800.0 PL=0
MOVL C01660 V=800.0 PL=0
MOVL C01661 V=800.0 PL=0
MOVL C01662 V=800.0 PL=0
MOVL C01663 V=800.0 PL=0
MOVL C01664 V=800.0 PL=0
MOVL C01665 V=800.0 PL=0
MOVL C01666 V=800.0 PL=0
MOVL C01667 V=800.0 PL=0
MOVL C01668 V=800.0 PL=0
MOVL C01669 V=800.0 PL=0
MOVL C01670 V=800.0 PL=0
MOVL C01671 V=800.0 PL=0
MOVL C01672 V=800.0 PL=0
MOVL C01673 V=800.0 PL=0
MOVL C01674 V=800.0 PL=0
MOVL C01675 V=800.0 PL=0
MOVL C01676 V=800.0 PL=0
MOVL C01677 V=800.0 PL=0
MOVL C01678 V=800.0 PL=0
MOVL C01679 V=800.0 PL=0
MOVL C01680 V=800.0 PL=0
MOVL C01681 V=800.0 PL=0
MOVL C01682 V=800.0 PL=0
MOVL C01683 V=800.0 PL=0
MOVL C01684 V=800.0 PL=0
MOVL C01685 V=800.0 PL=0
MOVL C01686 V=800.0 PL=0
MOVL C01687 V=800.0 PL=0
MOVL C01688 V=800.0 PL=0
MOVL C01689 V=800.0 PL=0
MOVL C01690 V=800.0 PL=0
MOVL C01691 V=800.0 PL=0
MOVL C01692 V=800.0 PL=0
MOVL C01693 V=800.0 PL=0
MOVL C01694 V=800.0 PL=0
MOVL C01695 V=800.0 PL=0
MOVL C01696 V=800.0 PL=0
MOVL C01697 V=800.0 PL=0
MOVL C01698 V=800.0 PL=0
MOVL C01699 V=800.0 PL=0
MOVL C01700 V=800.0 PL=0
MOVL C01701 V=800.0 PL=0
MOVL C01702 V=800.0 PL=0
MOVL C01703 V=800.0 PL=0
MOVL C01704 V=800.0 PL=0
MOVL C01705 V=800.0 PL=0
MOVL C01706 V=800.0 PL=0
MOVL C01707 V=800.0 PL=0
MOVL C01708 V=800.0 PL=0
MOVL C01709 V=800.0 PL=0
MOVL C01710 V=800.0 PL=0
MOVL C01711 V=800.0 PL=0
MOVL C01712 V=800.0 PL=0
MOVL C01713 V=800.0 PL=0
MOVL C01714 V=800.0 PL=0
MOVL C01715 V=800.0 PL=0
MOVL C01716 V=800.0 PL=0
MOVL C01717 V=800.0 PL=0
MOVL C01718 V=800.0 PL=0
MOVL C01719 V=800.0 PL=0
MOVL C01720 V=800.0 PL=0
MOVL C01721 V=800.0 PL=0
MOVL C01722 V=800.0 PL=0
MOVL C01723 V=800.0 PL=0
MOVL C01724 V=800.0 PL=0
MOVL C01725 V=800.0 PL=0
MOVL C01726 V=800.0 PL=0
MOVL C01727 V=800.0 PL=0
MOVL C01728 V=800.0 PL=0
MOVL C01729 V=800.0 PL=0
MOVL C01730 V=800.0 PL=0
MOVL C01731 V=800.0 PL=0
MOVL C01732 V=800.0 PL=0
MOVL C01733 V=800.0 PL=0
MOVL C01734 V=800.0 PL=0
MOVL C01735 V=800.0 PL=0
MOVL C01736 V=800.0 PL=0
MOVL C01737 V=800.0 PL=0
MOVL C01738 V=800.0 PL=0
MOVL C01739 V=800.0 PL=0
MOVL C01740 V=800.0 PL=0
MOVL C01741 V=800.0 PL=0
MOVL C01742 V=800.0 PL=0
MOVL C01743 V=800.0 PL=0
MOVL C01744 V=800.0 PL=0
MOVL C01745 V=800.0 PL=0
MOVL C01746 V=800.0 PL=0
MOVL C01747 V=800.0 PL=0
MOVL C01748 V=800.0 PL=0
MOVL C01749 V=800.0 PL=0
MOVL C01750 V=800.0 PL=0
MOVL C01751 V=800.0 PL=0
MOVL C01752 V=800.0 PL=0
MOVL C01753 V=800.0 PL=0
MOVL C01754 V=800.0 PL=0
MOVL C01755 V=800.0 PL=0
MOVL C01756 V=800.0 PL=0
MOVL C01757 V=800.0 PL=0
MOVL C01758 V=800.0 PL=0
MOVL C01759 V=800.0 PL=0
MOVL C01760 V=800.0 PL=0
MOVL C01761 V=800.0 PL=0
MOVL C01762 V=800.0 PL=0
MOVL C01763 V=800.0 PL=0
MOVL C01764 V=800.0 PL=0
MOVL C01765 V=800.0 PL=0
MOVL C01766 V=800.0 PL=0
MOVL C01767 V=800.0 PL=0
MOVL C01768 V=800.0 PL=0
MOVL C01769 V=800.0 PL=0
MOVL C01770 V=800.0 PL=0
MOVL C01771 V=800.0 PL=0
MOVL C01772 V=800.0 PL=0
MOVL C01773 V=800.0 PL=0
MOVL C01774 V=800.0 PL=0
MOVL C01775 V=800.0 PL=0
MOVL C01776 V=800.0 PL=0
MOVL C01777 V=800.0 PL=0
MOVL C01778 V=800.0 PL=0
MOVL C01779 V=800.0 PL=0
MOVL C01780 V=800.0 PL=0
MOVL C01781 V=800.0 PL=0
MOVL C01782 V=800.0 PL=0
MOVL C01783 V=800.0 PL=0
MOVL C01784 V=800.0 PL=0
MOVL C01785 V=800.0 PL=0
MOVL C01786 V=800.0 PL=0
MOVL C01787 V=800.0 PL=0
MOVL C01788 V=800.0 PL=0
MOVL C01789 V=800.0 PL=0
MOVL C01790 V=800.0 PL=0
MOVL C01791 V=800.0 PL=0
MOVL C01792 V=800.0 PL=0
MOVL C01793 V=800.0 PL=0
MOVL C01794 V=800.0 PL=0
MOVL C01795 V=800.0 PL=0
MOVL C01796 V=800.0 PL=0
MOVL C01797 V=800.0 PL=0
MOVL C01798 V=800.0 PL=0
MOVL C01799 V=800.0 PL=0
MOVL C01800 V=800.0 PL=0
MOVL C01801 V=800.0 PL=0
MOVL C01802 V=800.0 PL=0
MOVL C01803 V=800.0 PL=0
MOVL C01804 V=800.0 PL=0
MOVL C01805 V=800.0 PL=0
MOVL C01806 V=800.0 PL=0
MOVL C01807 V=800.0 PL=0
MOVL C01808 V=800.0 PL=0
MOVL C01809 V=800.0 PL=0
MOVL C01810 V=800.0 PL=0
MOVL C01811 V=800.0 PL=0
MOVL C01812 V=800.0 PL=0
MOVL C01813 V=800.0 PL=0
MOVL C01814 V=800.0 PL=0
MOVL C01815 V=800.0 PL=0
MOVL C01816 V=800.0 PL=0
MOVL C01817 V=800.0 PL=0
MOVL C01818 V=800.0 PL=0
MOVL C01819 V=800.0 PL=0
MOVL C01820 V=800.0 PL=0
MOVL C01821 V=800.0 PL=0
MOVL C01822 V=800.0 PL=0
MOVL C01823 V=800.0 PL=0
MOVL C01824 V=800.0 PL=0
MOVL C01825 V=800.0 PL=0
MOVL C01826 V=800.0 PL=0
MOVL C01827 V=800.0 PL=0
MOVL C01828 V=800.0 PL=0
MOVL C01829 V=800.0 PL=0
MOVL C01830 V=800.0 PL=0
MOVL C01831 V=800.0 PL=0
MOVL C01832 V=800.0 PL=0
MOVL C01833 V=800.0 PL=0
MOVL C01834 V=800.0 PL=0
MOVL C01835 V=800.0 PL=0
MOVL C01836 V=800.0 PL=0
MOVL C01837 V=800.0 PL=0
MOVL C01838 V=800.0 PL=0
MOVL C01839 V=800.0 PL=0
MOVL C01840 V=800.0 PL=0
MOVL C01841 V=800.0 PL=0
MOVL C01842 V=800.0 PL=0
MOVL C01843 V=800.0 PL=0
MOVL C01844 V=800.0 PL=0
MOVL C01845 V=800.0 PL=0
MOVL C01846 V=800.0 PL=0
MOVL C01847 V=800.0 PL=0
MOVL C01848 V=800.0 PL=0
MOVL C01849 V=800.0 PL=0
MOVL C01850 V=800.0 PL=0
MOVL C01851 V=800.0 PL=0
MOVL C01852 V=800.0 PL=0
MOVL C01853 V=800.0 PL=0
MOVL C01854 V=800.0 PL=0
MOVL C01855 V=800.0 PL=0
MOVL C01856 V=800.0 PL=0
MOVL C01857 V=800.0 PL=0
MOVL C01858 V=800.0 PL=0
MOVL C01859 V=800.0 PL=0
MOVL C01860 V=800.0 PL=0
MOVL C01861 V=800.0 PL=0
MOVL C01862 V=800.0 PL=0
MOVL C01863 V=800.0 PL=0
MOVL C01864 V=800.0 PL=0
MOVL C01865 V=800.0 PL=0
MOVL C01866 V=800.0 PL=0
MOVL C01867 V=800.0 PL=0
MOVL C01868 V=800.0 PL=0
MOVL C01869 V=800.0 PL=0
MOVL C01870 V=800.0 PL=0
MOVL C01871 V=800.0 PL=0
MOVL C01872 V=800.0 PL=0
MOVL C01873 V=800.0 PL=0
MOVL C01874 V=800.0 PL=0
MOVL C01875 V=800.0 PL=0
MOVL C01876 V=800.0 PL=0
MOVL C01877 V=800.0 PL=0
MOVL C01878 V=800.0 PL=0
MOVL C01879 V=800.0 PL=0
MOVL C01880 V=800.0 PL=0
MOVL C01881 V=800.0 PL=0
MOVL C01882 V=800.0 PL=0
MOVL C01883 V=800.0 PL=0
MOVL C01884 V=800.0 PL=0
MOVL C01885 V=800.0 PL=0
MOVL C01886 V=800.0 PL=0
MOVL C01887 V=800.0 PL=0
MOVL C01888 V=800.0 PL=0
MOVL C01889 V=800.0 PL=0
MOVL C01890 V=800.0 PL=0
MOVL C01891 V=800.0 PL=0
MOVL C01892 V=800.0 PL=0
MOVL C01893 V=800.0 PL=0
MOVL C01894 V=800.0 PL=0
MOVL C01895 V=800.0 PL=0
MOVL C01896 V=800.0 PL=0
MOVL C01897 V=800.0 PL=0
MOVL C01898 V=800.0 PL=0
MOVL C01899 V=800.0 PL=0
MOVL C01900 V=800.0 PL=0
MOVL C01901 V=800.0 PL=0
MOVL C01902 V=800.0 PL=0
MOVL C01903 V=800.0 PL=0
MOVL C01904 V=800.0 PL=0
MOVL C01905 V=800.0 PL=0
MOVL C01906 V=800.0 PL=0
MOVL C01907 V=800.0 PL=0
MOVL C01908 V=800.0 PL=0
MOVL C01909 V=800.0 PL=0
MOVL C01910 V=800.0 PL=0
MOVL C01911 V=800.0 PL=0
MOVL C01912 V=800.0 PL=0
MOVL C01913 V=800.0 PL=0
MOVL C01914 V=800.0 PL=0
MOVL C01915 V=800.0 PL=0
MOVL C01916 V=800.0 PL=0
MOVL C01917 V=800.0 PL=0
MOVL C01918 V=800.0 PL=0
MOVL C01919 V=800.0 PL=0
MOVL C01920 V=800.0 PL=0
MOVL C01921 V=800.0 PL=0
MOVL C01922 V=800.0 PL=0
MOVL C01923 V=800.0 PL=0
MOVL C01924 V=800.0 PL=0
MOVL C01925 V=800.0 PL=0
MOVL C01926 V=800.0 PL=0
MOVL C01927 V=800.0 PL=0
MOVL C01928 V=800.0 PL=0
MOVL C01929 V=800.0 PL=0
MOVL C01930 V=800.0 PL=0
MOVL C01931 V=800.0 PL=0
MOVL C01932 V=800.0 PL=0
MOVL C01933 V=800.0 PL=0
MOVL C01934 V=800.0 PL=0
MOVL C01935 V=800.0 PL=0
MOVL C01936 V=800.0 PL=0
MOVL C01937 V=800.0 PL=0
MOVL C01938 V=800.0 PL=0
MOVL C01939 V=800.0 PL=0
MOVL C01940 V=800.0 PL=0
MOVL C01941 V=800.0 PL=0
MOVL C01942 V=800.0 PL=0
MOVL C01943 V=800.0 PL=0
MOVL C01944 V=800.0 PL=0
MOVL C01945 V=800.0 PL=0
MOVL C01946 V=800.0 PL=0
MOVL C01947 V=800.0 PL=0
MOVL C01948 V=800.0 PL=0
MOVL C01949 V=800.0 PL=0
MOVL C01950 V=800.0 PL=0
MOVL C01951 V=800.0 PL=0
MOVL C01952 V=800.0 PL=0
MOVL C01953 V=800.0 PL=0
MOVL C01954 V=800.0 PL=0
MOVL C01955 V=800.0 PL=0
MOVL C01956 V=800.0 PL=0
MOVL C01957 V=800.0 PL=0
MOVL C01958 V=800.0 PL=0
MOVL C01959 V=800.0 PL=0
MOVL C01960 V=800.0 PL=0
MOVL C01961 V=800.0 PL=0
MOVL C01962 V=800.0 PL=0
MOVL C01963 V=800.0 PL=0
MOVL C01964 V=800.0 PL=0
MOVL C01965 V=800.0 PL=0
MOVL C01966 V=800.0 PL=0
MOVL C01967 V=800.0 PL=0
MOVL C01968 V=800.0 PL=0
MOVL C01969 V=800.0 PL=0
MOVL C01970 V=800.0 PL=0
MOVL C01971 V=800.0 PL=0
MOVL C01972 V=800.0 PL=0
MOVL C01973 V=800.0 PL=0
MOVL C01974 V=800.0 PL=0
MOVL C01975 V=800.0 PL=0
MOVL C01976 V=800.0 PL=0
MOVL C01977 V=800.0 PL=0
MOVL C01978 V=800.0 PL=0
MOVL C01979 V=800.0 PL=0
MOVL C01980 V=800.0 PL=0
MOVL C01981 V=800.0 PL=0
MOVL C01982 V=800.0 PL=0
MOVL C01983 V=800.0 PL=0
MOVL C01984 V=800.0 PL=0
MOVL C01985 V=800.0 PL=0
MOVL C01986 V=800.0 PL=0
MOVL C01987 V=800.0 PL=0
MOVL C01988 V=800.0 PL=0
MOVL C01989 V=800.0 PL=0
MOVL C01990 V=800.0 PL=0
MOVL C01991 V=800.0 PL=0
MOVL C01992 V=800.0 PL=0
MOVL C01993 V=800.0 PL=0
MOVL C01994 V=800.0 PL=0
MOVL C01995 V=800.0 PL=0
MOVL C01996 V=800.0 PL=0
MOVL C01997 V=800.0 PL=0
MOVL C01998 V=800.0 PL=0
MOVL C01999 V=800.0 PL=0
MOVL C02000 V=800.0 PL=0
MOVL C02001 V=800.0 PL=0
MOVL C02002 V=800.0 PL=0
MOVL C02003 V=800.0 PL=0
MOVL C02004 V=800.0 PL=0
MOVL C02005 V=800.0 PL=0
MOVL C02006 V=800.0 PL=0
MOVL C02007 V=800.0 PL=0
MOVL C02008 V=800.0 PL=0
MOVL C02009 V=800.0 PL=0
MOVL C02010 V=800.0 PL=0
MOVL C02011 V=800.0 PL=0
MOVL C02012 V=800.0 PL=0
MOVL C02013 V=800.0 PL=0
MOVL C02014 V=800.0 PL=0
MOVL C02015 V=800.0 PL=0
MOVL C02016 V=800.0 PL=0
MOVL C02017 V=800.0 PL=0
MOVL C02018 V=800.0 PL=0
MOVL C02019 V=800.0 PL=0
MOVL C02020 V=800.0 PL=0
MOVL C02021 V=800.0 PL=0
MOVL C02022 V=800.0 PL=0
MOVL C02023 V=800.0 PL=0
MOVL C02024 V=800.0 PL=0
MOVL C02025 V=800.0 PL=0
MOVL C02026 V=800.0 PL=0
MOVL C02027 V=800.0 PL=0
MOVL C02028 V=800.0 PL=0
MOVL C02029 V=800.0 PL=0
MOVL C02030 V=800.0 PL=0
MOVL C02031 V=800.0 PL=0
MOVL C02032 V=800.0 PL=0
MOVL C02033 V=800.0 PL=0
MOVL C02034 V=800.0 PL=0
MOVL C02035 V=800.0 PL=0
MOVL C02036 V=800.0 PL=0
MOVL C02037 V=800.0 PL=0
MOVL C02038 V=800.0 PL=0
MOVL C02039 V=800.0 PL=0
MOVL C02040 V=800.0 PL=0
MOVL C02041 V=800.0 PL=0
MOVL C02042 V=800.0 PL=0
MOVL C02043 V=800.0 PL=0
MOVL C02044 V=800.0 PL=0
MOVL C02045 V=800.0 PL=0
MOVL C02046 V=800.0 PL=0
MOVL C02047 V=800.0 PL=0
MOVL C02048 V=800.0 PL=0
MOVL C02049 V=800.0 PL=0
MOVL C02050 V=800.0 PL=0
MOVL C02051 V=800.0 PL=0
MOVL C02052 V=800.0 PL=0
MOVL C02053 V=800.0 PL=0
MOVL C02054 V=800.0 PL=0
MOVL C02055 V=800.0 PL=0
MOVL C02056 V=800.0 PL=0
MOVL C02057 V=800.0 PL=0
MOVL C02058 V=800.0 PL=0
MOVL C02059 V=800.0 PL=0
MOVL C02060 V=800.0 PL=0
MOVL C02061 V=800.0 PL=0
MOVL C02062 V=800.0 PL=0
MOVL C02063 V=800.0 PL=0
MOVL C02064 V=800.0 PL=0
MOVL C02065 V=800.0 PL=0
MOVL C02066 V=800.0 PL=0
MOVL C02067 V=800.0 PL=0
MOVL C02068 V=800.0 PL=0
MOVL C02069 V=800.0 PL=0
MOVL C02070 V=800.0 PL=0
MOVL C02071 V=800.0 PL=0
MOVL C02072 V=800.0 PL=0
MOVL C02073 V=800.0 PL=0
MOVL C02074 V=800.0 PL=0
MOVL C02075 V=800.0 PL=0
MOVL C02076 V=800.0 PL=0
MOVL C02077 V=800.0 PL=0
MOVL C02078 V=800.0 PL=0
MOVL C02079 V=800.0 PL=0
MOVL C02080 V=800.0 PL=0
MOVL C02081 V=800.0 PL=0
MOVL C02082 V=800.0 PL=0
MOVL C02083 V=800.0 PL=0
MOVL C02084 V=800.0 PL=0
MOVL C02085 V=800.0 PL=0
MOVL C02086 V=800.0 PL=0
MOVL C02087 V=800.0 PL=0
MOVL C02088 V=800.0 PL=0
MOVL C02089 V=800.0 PL=0
MOVL C02090 V=800.0 PL=0
MOVL C02091 V=800.0 PL=0
MOVL C02092 V=800.0 PL=0
MOVL C02093 V=800.0 PL=0
MOVL C02094 V=800.0 PL=0
MOVL C02095 V=800.0 PL=0
MOVL C02096 V=800.0 PL=0
MOVL C02097 V=800.0 PL=0
MOVL C02098 V=800.0 PL=0
MOVL C02099 V=800.0 PL=0
MOVL C02100 V=800.0 PL=0
MOVL C02101 V=800.0 PL=0
MOVL C02102 V=800.0 PL=0
MOVL C02103 V=800.0 PL=0
MOVL C02104 V=800.0 PL=0
MOVL C02105 V=800.0 PL=0
MOVL C02106 V=800.0 PL=0
MOVL C02107 V=800.0 PL=0
MOVL C02108 V=800.0 PL=0
MOVL C02109 V=800.0 PL=0
MOVL C02110 V=800.0 PL=0
MOVL C02111 V=800.0 PL=0
MOVL C02112 V=800.0 PL=0
MOVL C02113 V=800.0 PL=0
MOVL C02114 V=800.0 PL=0
MOVL C02115 V=800.0 PL=0
MOVL C02116 V=800.0 PL=0
MOVL C02117 V=800.0 PL=0
MOVL C02118 V=800.0 PL=0
MOVL C02119 V=800.0 PL=0
MOVL C02120 V=800.0 PL=0
MOVL C02121 V=800.0 PL=0
MOVL C02122 V=800.0 PL=0
MOVL C02123 V=800.0 PL=0
